FUNCTION_BLOCK "Blok_Jazdy_Band"	// FB 5
VERSION : 0.1
VAR
  Banda_1 : FB 30;
  Banda_2 : FB 30;
  Banda_3 : FB 30;
  Banda_4 : FB 31;
  Banda_5 : FB 30;
  Banda_6 : FB 30;
  Banda_7 : FB 30;
  Banda_8 : FB 30;
  Banda_9 : FB 30;
  Banda_12 : FB 30;
  Banda_13 : FB 32;
  Banda_14 : FB 30;
END_VAR
BEGIN
NETWORK
TITLE =
//Ten network celowo jest wolny
NETWORK
TITLE =
//Opoznienie wlotu bandy 1
//Uwaga Stare !!!
//      CALL  "Opoznienie_Wlotu"
//       Wejscie :="AIO".Banda_1.Foto_1
//       Timmer_1:=T12
//       Timmer_2:=T13
//       Wyjscie :="M_Foto_1_Banda_1"
//       Zmienna :="Help_M_40_3"
NETWORK
TITLE =
//Banda 1
//Uwaga Stare !!!
//      CALL  #Banda_1
//       S_Marka_Bezpieczenstwa :="Marka_Bezpieczenstwa"
//       i_Foto_Koniec          :="M_Foto_1_Banda_1"
//       i_Zez_Od_Nast          :="AIO".Banda_2.Zez_Do_Pop
//       i_Paleta_Dost_Od_Nast  :="AIO".Banda_2.Paleta_Dost_do_Pop
//       i_Zabierz_Od_Pop       :=
//       Czas_Kontroli_Przejazdu:=T#10S
//       o_Zabierz_Do_Nast      :="AIO".Banda_1.Zabierz_do_Nast
//       o_Zez_Do_Pop           :="AIO".Banda_1.Zez_Do_Pop
//       o_Paleta_Dost_do_Pop   :="AIO".Banda_1.Paleta_Dost_do_Pop
//       o_Motor_Lewo           :="AIO".Banda_1.C_Wise
NETWORK
TITLE =
//Banda 2. Uznawana za Wlot 1
//Uwaga Stare !!!
//      CALL  #Banda_2
//       S_Marka_Bezpieczenstwa :="Marka_Bezpieczenstwa"
//       i_Foto_Koniec          :="AIO".Banda_2.Foto_1
//       i_Zez_Od_Nast          :="AIO".Banda_4.Zez_Do_Pop_Wlot_1
//       i_Paleta_Dost_Od_Nast  :="AIO".Banda_4.Potw_Dost_Wlot_1
//       i_Zabierz_Od_Pop       :="AIO".Banda_1.Zabierz_do_Nast
//       Czas_Kontroli_Przejazdu:=T#10S
//       o_Zabierz_Do_Nast      :="AIO".Banda_2.Zabierz_do_Nast
//       o_Zez_Do_Pop           :="AIO".Banda_2.Zez_Do_Pop
//       o_Paleta_Dost_do_Pop   :="AIO".Banda_2.Paleta_Dost_do_Pop
//       o_Motor_Lewo           :="AIO".Banda_2.C_Wise
NETWORK
TITLE =
//Opoznienie wlotu banda 3
      CALL  "Opoznienie_Wlotu" (
           Wejscie                  := "AIO".Banda_3.Foto_1,
           Timmer_1                 := T 14,
           Timmer_2                 := T 15,
           Wyjscie                  := "M_Foto_1_Banda_3",
           Zmienna                  := "Help_M_40_5");
NETWORK
TITLE =
//Banda 3. Uznawana za Wlot 2
      CALL  #Banda_3 (
           S_Marka_Bezpieczenstwa   := "Marka_Bezpieczenstwa",
           i_Foto_Koniec            := "M_Foto_1_Banda_3",
           i_Zez_Od_Nast            := DIX 7.2,
           i_Paleta_Dost_Od_Nast    := DIX 7.3,
           Czas_Kontroli_Przejazdu  := T#10S,
           o_Zabierz_Do_Nast        := DIX 5.2,
           o_Zez_Do_Pop             := DIX 5.0,
           o_Paleta_Dost_do_Pop     := DIX 5.1,
           o_Motor_Lewo             := DIX 4.4);
NETWORK
TITLE =
//Banda 4 obrotowa
      CALL  #Banda_4 (
           i_Marka_bezpieczenstwa   := "Marka_Bezpieczenstwa",
           i_Foto_1                 := DIX 6.2,
           i_Foto_2                 := DIX 6.3,
           i_Zez_od_Nast            := DIX 9.0,
           i_Zabierz_od_Wlot_1      := DIX 3.2,
           i_Zabierz_od_Wlot_2      := DIX 5.2,
           i_Paleta_Odb_Wylot       := DIX 9.1,
           i_czuj_poz_Wlot_1        := DIX 36.3,
           i_czuj_ham_Wlot_1        := DIX 36.2,
           i_czuj_poz_Wlot_2        := DIX 36.0,
           i_czuj_ham_Wlot_2        := DIX 36.1,
           i_Foto_Wlot_1            := "M_Foto_1_Banda_2",
           i_Foto_Wlot_2            := "M_Foto_1_Banda_3",
           o_Zez_do_Wlot_1          := DIX 7.0,
           o_Zez_do_Wlot_2          := DIX 7.2,
           o_Paleta_Dost_Wlot_1     := DIX 7.1,
           o_Paleta_Dost_Wlot_2     := DIX 7.3,
           o_Zabierz_do_Nast        := DIX 7.4,
           o_Motor_1_lewo           := DIX 6.4,
           o_Motor_1_prawo          := DIX 6.5,
           o_Motor_2_obr_s_Wlot_1   := DIX 34.5,
           o_Motor_2_obr_s_Wlot_2   := DIX 34.4,
           o_Motor_2_Wolno          := DIX 34.6);
NETWORK
TITLE =
//Banda 5
      CALL  #Banda_5 (
           S_Marka_Bezpieczenstwa   := "Marka_Bezpieczenstwa",
           i_Foto_Koniec            := DIX 8.2,
           i_Zez_Od_Nast            := DIX 11.0,
           i_Paleta_Dost_Od_Nast    := DIX 11.1,
           i_Zabierz_Od_Pop         := DIX 7.4,
           Czas_Kontroli_Przejazdu  := T#10S,
           o_Zabierz_Do_Nast        := DIX 9.2,
           o_Zez_Do_Pop             := DIX 9.0,
           o_Paleta_Dost_do_Pop     := DIX 9.1,
           o_Motor_Lewo             := DIX 8.4);
NETWORK
TITLE =
//Banda 6
      CALL  #Banda_6 (
           S_Marka_Bezpieczenstwa   := "Marka_Bezpieczenstwa",
           i_Foto_Koniec            := DIX 10.2,
           i_Zez_Od_Nast            := DIX 13.0,
           i_Paleta_Dost_Od_Nast    := DIX 13.1,
           i_Zabierz_Od_Pop         := DIX 9.2,
           Czas_Kontroli_Przejazdu  := T#10S,
           o_Zabierz_Do_Nast        := DIX 11.2,
           o_Zez_Do_Pop             := DIX 11.0,
           o_Paleta_Dost_do_Pop     := DIX 11.1,
           o_Motor_Lewo             := DIX 10.4);
NETWORK
TITLE =
//Banda 7
      CALL  #Banda_7 (
           S_Marka_Bezpieczenstwa   := "Marka_Bezpieczenstwa",
           i_Foto_Koniec            := DIX 12.2,
           i_Zez_Od_Nast            := DIX 15.0,
           i_Paleta_Dost_Od_Nast    := DIX 15.1,
           i_Zabierz_Od_Pop         := DIX 11.2,
           Czas_Kontroli_Przejazdu  := T#10S,
           o_Zabierz_Do_Nast        := DIX 13.2,
           o_Zez_Do_Pop             := DIX 13.0,
           o_Paleta_Dost_do_Pop     := DIX 13.1,
           o_Motor_Lewo             := DIX 12.4);
NETWORK
TITLE =
//Banda 8
      CALL  #Banda_8 (
           S_Marka_Bezpieczenstwa   := "Marka_Bezpieczenstwa",
           i_Foto_Koniec            := DIX 14.2,
           i_Zez_Od_Nast            := DIX 17.0,
           i_Paleta_Dost_Od_Nast    := DIX 17.1,
           i_Zabierz_Od_Pop         := DIX 13.2,
           Czas_Kontroli_Przejazdu  := T#10S,
           o_Zabierz_Do_Nast        := DIX 15.2,
           o_Zez_Do_Pop             := DIX 15.0,
           o_Paleta_Dost_do_Pop     := DIX 15.1,
           o_Motor_Lewo             := DIX 14.4);
NETWORK
TITLE =
//Banda 9
      CALL  #Banda_9 (
           S_Marka_Bezpieczenstwa   := "Marka_Bezpieczenstwa",
           i_Foto_Koniec            := DIX 16.2,
           i_Zez_Od_Nast            := DIX 19.0,
           i_Paleta_Dost_Od_Nast    := DIX 19.1,
           i_Zabierz_Od_Pop         := DIX 15.2,
           Czas_Kontroli_Przejazdu  := T#10S,
           o_Zabierz_Do_Nast        := DIX 17.2,
           o_Zez_Do_Pop             := DIX 17.0,
           o_Paleta_Dost_do_Pop     := DIX 17.1,
           o_Motor_Lewo             := DIX 16.4);
NETWORK
TITLE = Zezwolenie do poprzedniej
//Banda 10 to foliarka. Tu jest interface laczacy dwie maszyny
      A     "MPI_GD".IN.Zezwolenie_Na_Wjazd_10;
      =     "AIO".Banda_10.Zez_Do_Pop;
//---
      A     "MPI_GD".IN.Potw_Dost_Na_Wjazd_10;
      =     "AIO".Banda_10.Paleta_Dost_do_Pop;
      A     "AIO".Banda_9.Zabierz_do_Nast;
      =     "MPI_GD".OUT.Zabierz_Na_Bande_10;
NETWORK
TITLE =
//Banda 11 to wylot z foliarki. Tu jest interface laczacy.Uwazana jako wlot 1
      A     "AIO".Banda_13.Zez_Do_Pop_Wlot_1;
      =     "MPI_GD".OUT.Zezwolenie_Na_Wyjazd_11;
//Przedluzenine czasu trwania sygnalu potwierdzenia
      A     "AIO".Banda_13.Potw_Dost_Wlot_1;
      L     S5T#200MS;
      SE    T 20;
      A     T 20;
      =     "MPI_GD".OUT.Potw_Dost_Na_Wyjazd_11;
//Przejecie palety
      A     "MPI_GD".IN.Zabierz_Na_Bande_11;
      =     "AIO".Banda_11.Zabierz_do_Nast;
      A     "MPI_GD".IN.Paleta_Obecna_Na_7_Tr;
      =     "M_Foto_1_Banda_11";
      A     "AIO".Czuj_21.Czujnik_90_St;
      AN    "AIO".Czuj_21.Czujnik_0_St;
      AN    "AIO".Czuj_22.Czujnik_45_St_CW;
      AN    "AIO".Czuj_22.Czujnik_45_St_CCW;
      =     "MPI_GD".OUT.Obrot_Na_Poz_Wlot_1;
NETWORK
TITLE =
//Opoznienie wlotu 2 przy obrotnicy 2
      CALL  "Opoznienie_Wlotu" (
           Wejscie                  := "AIO".Banda_12.Foto_1,
           Timmer_1                 := T 16,
           Timmer_2                 := T 17,
           Wyjscie                  := "M_Foto_1_Banda_12",
           Zmienna                  := "Help_M_40_7");
NETWORK
TITLE =
//Banda 12. Uwazana jako wlot 2.
      CALL  #Banda_12 (
           S_Marka_Bezpieczenstwa   := "Marka_Bezpieczenstwa",
           i_Foto_Koniec            := "M_Foto_1_Banda_12",
           i_Zez_Od_Nast            := DIX 25.2,
           i_Paleta_Dost_Od_Nast    := DIX 25.3,
           Czas_Kontroli_Przejazdu  := T#10S,
           o_Zabierz_Do_Nast        := DIX 23.2,
           o_Zez_Do_Pop             := DIX 23.0,
           o_Paleta_Dost_do_Pop     := DIX 23.1,
           o_Motor_Lewo             := DIX 22.4);
NETWORK
TITLE =
//banda 13 obrotowa
      CALL  #Banda_13 (
           i_Marka_bezpieczenstwa   := "Marka_Bezpieczenstwa",
           i_Foto_1                 := DIX 24.2,
           i_Foto_2                 := DIX 24.3,
           i_Zez_od_Nast            := DIX 27.0,
           i_Zabierz_od_Wlot_1      := DIX 21.2,
           i_Zabierz_od_Wlot_2      := DIX 23.2,
           i_Paleta_Odb_Wylot       := DIX 27.1,
           i_czuj_poz_Wlot_1        := DIX 40.3,
           i_czuj_ham_Wlot_1        := DIX 40.2,
           i_czuj_poz_Wlot_2        := DIX 40.0,
           i_czuj_ham_Wlot_2        := DIX 40.1,
           i_Czuj_poz_45_deg        := DIX 42.0,
           i_Czuj_ham_45_deg        := DIX 42.1,
           i_Foto_Wlot_1            := "M_Foto_1_Banda_11",
           i_Foto_Wlot_2            := "M_Foto_1_Banda_12",
           i_Etyk_praca_wlacz       := "Praca_Z_Etykietami",
           i_Etyk_poz_podst         := "Silownik_Etyk_Tyl",
           i_Etyk_obraz_w_pamieci   := "Dane_W_Drukarce",
           i_Etyk_syg_gotowosci     := "Etyk_Gotowa",
           i_Etyk_brak_materialu    := "Brak_Papieru",
           i_Etyk_Przycisk_Drukuj   := "Drukuj_Recznie",
           o_Zez_do_Wlot_1          := DIX 25.0,
           o_Zez_do_Wlot_2          := DIX 25.2,
           o_Paleta_Dost_Wlot_1     := DIX 25.1,
           o_Paleta_Dost_Wlot_2     := DIX 25.3,
           o_Zabierz_do_Nast        := DIX 25.4,
           o_Motor_1_lewo           := DIX 24.4,
           o_Motor_1_prawo          := DIX 24.5,
           o_Motor_2_obr_s_Wlot_1   := DIX 38.5,
           o_Motor_2_obr_s_Wlot_2   := DIX 38.4,
           o_Motor_2_Wolno          := DIX 38.6,
           o_Silownik_etykiety      := "Silownik_Etykiet",
           o_Drukuj_Etykiete        := "Drukuj_Etykiete",
           o_Zalaczenie_Skanera     := "Zalacz_Skaner",
           o_Lampka_Przycisk_Drukuj := "Lampka_Obraz_W_Pamieci");
NETWORK
TITLE =
//Wywolanie opoznienia zatrzymania fotokomorki po wyjsciu z obrotnicy
      CALL  "Opoznienie_Wylotu" (
           Wejscie                  := "AIO".Banda_14.Foto_1,
           Timmer_1                 := T 10,
           Timmer_2                 := T 11,
           Wyjscie                  := "M_Foto_1_Banda_14",
           Zmienna                  := "Help_M_40_1");
NETWORK
TITLE =
//Banda 14.Banda uwazana jako wylot z obrotnicy.
      CALL  #Banda_14 (
           S_Marka_Bezpieczenstwa   := "Marka_Bezpieczenstwa",
           i_Foto_Koniec            := "M_Foto_1_Banda_14",
           i_Zabierz_Od_Pop         := DIX 25.4,
           Czas_Kontroli_Przejazdu  := T#10S,
           o_Zabierz_Do_Nast        := DIX 27.2,
           o_Zez_Do_Pop             := DIX 27.0,
           o_Paleta_Dost_do_Pop     := DIX 27.1,
           o_Motor_Lewo             := DIX 26.4);
//      SET   
//      S     "Zalacz_Skaner"
END_FUNCTION_BLOCK

FUNCTION_BLOCK "Filtr_zbocza_2"	// FB 14
//Funkcja wykrywajace zbocze fotokomorki uwzgledniajaca nieczu³osc elementu
//
AUTHOR : Kng
FAMILY : Fun
NAME : Zb_1
VERSION : 0.1
VAR_INPUT
  Foto : BOOL ;
END_VAR
VAR_OUTPUT
  pos_zbocze : BOOL ;
END_VAR
VAR
  Opoz_zbocza_pos : SFB 4;
  p_Sygnal_foto : BOOL ;
  b_Opoz_poz : BOOL ;
  Help_zb_poz : BOOL ;
END_VAR
BEGIN
NETWORK
TITLE =
      CALL  #Opoz_zbocza_pos (
           IN                       := #Foto,
           PT                       := T#100MS,
           Q                        := #b_Opoz_poz);
      A     #b_Opoz_poz;
      S     #p_Sygnal_foto;
      AN    #Foto;
      R     #p_Sygnal_foto;
      A     #p_Sygnal_foto;
      FP    #Help_zb_poz;
      =     #pos_zbocze;
      BEU;
END_FUNCTION_BLOCK

FUNCTION_BLOCK "T_ON"	// FB 20
//Funkcja zatrzymujaca czas gdy na wejsciu stop pojawi sie stan niski. Wartosc 
//wejscia TON nie jest wtedy brana pod uwage. 
AUTHOR : Kng
NAME : Help_FB
VERSION : 0.1
VAR_INPUT
  IN : BOOL ;	//Wejscie aktywujace timer
  STOP : BOOL ;	//Sygnal aktywny stanem wysokim
  PT : TIME ;	//Czas zadany
END_VAR
VAR_OUTPUT
  Q_0 : BOOL ;
END_VAR
VAR_IN_OUT
  ET : TIME ;
END_VAR
VAR
  T_1 : SFB 4;
  Help_Zbocze_1 : BOOL ;
  Help_Zbocze_2 : BOOL ;
  Help_Zbocze_3 : BOOL ;
END_VAR
BEGIN
NETWORK
TITLE =
//Ten network celowo jest wolny
NETWORK
TITLE =
// Zapisanie wartosci czasu w pamieci
      A     #STOP;
      FN    #Help_Zbocze_1;
      A     #IN;
      JCN   et_1;
      L     #T_1.PT;
      L     #T_1.ET;
      -D;
      T     #T_1.PT;
      SET;
      R     #T_1.IN;
et_1: NOP   0;
//Przywrocenie czasu zapisanego
      A     #STOP;
      FP    #Help_Zbocze_2;
      A     #IN;
      S     #T_1.IN;
//Warunki poczatkowe
      A     #IN;
      FP    #Help_Zbocze_3;
      A     #STOP;
      JCN   et_3;
      L     #PT;
      T     #T_1.PT;
      SET;
      S     #T_1.IN;
et_3: NOP   0;
//Wywolaj funkcje timera
      CALL  #T_1;
      A     #T_1.Q;
      S     #Q_0;
      AN    #IN;
      A     #STOP;
//Wystaw wyjscie gdy skonczy sie czas
      R     #T_1.IN;
      R     #Q_0;
      L     #T_1.PT;
      L     #T_1.ET;
      -D;
      T     #ET;
//Pokaz wartosc czasu
END_FUNCTION_BLOCK

FUNCTION_BLOCK "T_ON_+_RESET"	// FB 21
//Funkcja zatrzymujaca czas gdy na wejsciu stop pojawi sie stan niski. Wartosc 
//wejscia TON nie jest wtedy brana pod uwage. 
//Dodano przycisk reset.
AUTHOR : Kng
NAME : Help_FB
VERSION : 1.1
VAR_INPUT
  IN : BOOL ;	//Wejscie aktywujace timer
  STOP : BOOL ;	//Sygnal aktywny stanem wysokim
  PT : TIME ;	//Czas zadany
  RESET : BOOL ;	//Wejescie resetujace aktywne stanem wysokim
END_VAR
VAR_OUTPUT
  Q_0 : BOOL ;
END_VAR
VAR_IN_OUT
  ET : TIME ;
END_VAR
VAR
  T_1 : SFB 4;
  Help_Zbocze_1 : BOOL ;
  Help_Zbocze_2 : BOOL ;
  Help_Zbocze_3 : BOOL ;
  Help_Zbocze_4 : BOOL ;
  Help_Zbocze_5 : BOOL ;
END_VAR
BEGIN
NETWORK
TITLE =
//Ten network celowo jest wolny
NETWORK
TITLE =
      A     #RESET;
      S     #Help_Zbocze_4;
// Zapisanie wartosci czasu w pamieci
      A     #STOP;
      FN    #Help_Zbocze_1;
      A     #IN;
      JCN   et_2;
      L     #T_1.PT;
      L     #T_1.ET;
      -D;
      T     #T_1.PT;
      SET;
      R     #T_1.IN;
et_2: NOP   0;
//Przywrocenie czasu zapisanego
      A     #STOP;
      FP    #Help_Zbocze_2;
      A     #IN;
      S     #T_1.IN;
//Wystaw wyjscie gdy skonczy sie czas
      A     #T_1.Q;
      S     #Q_0;
      AN    #IN;
      A     #STOP;
      O;
      A     #RESET;
      R     #T_1.IN;
      R     #Q_0;
//Warunki poczatkowe  oraz reset
      AN    #RESET;
      A     #Help_Zbocze_4;
      O;
      A(;
      A     #IN;
      FP    #Help_Zbocze_3;
      A     #STOP;
      );
      JCN   et_3;
      L     #PT;
      T     #T_1.PT;
      SET;
      R     #Help_Zbocze_4;
//brak wysterownia jezeli reset robiony bez stopu
      A     #STOP;
      S     #T_1.IN;
et_3: NOP   0;
//Wywolaj funkcje timera
      CALL  #T_1;
      L     #T_1.PT;
      L     #T_1.ET;
      -D;
      T     #ET;
//Pokaz wartosc czasu
END_FUNCTION_BLOCK

FUNCTION_BLOCK "Banda_Podwojna"	// FB 29
//Funkcja realizujaca koncepcje bandy podwojnej:
//-pojedynczy silnik
//-2 fotokomorki
//
AUTHOR : Kng
FAMILY : Bandy
NAME : B_dual
VERSION : 0.3
VAR_INPUT
  S_Marka_Bezpieczenstwa : BOOL ;
  i_Foto_Srodek : BOOL ;	//Foto na srodku tasmy
  i_Foto_Koniec : BOOL ;	//Foto na koncu tasmy
  i_Zez_Od_Nast : BOOL ;
  i_Paleta_Dost_Od_Nast : BOOL ;
  i_Zabierz_Od_Pop : BOOL ;
  Czas_Kontroli_Przejazdu : TIME ;
END_VAR
VAR_OUTPUT
  o_Zabierz_Do_Nast : BOOL ;	//Rozkaz pobrania do nast bandy
  o_Zez_Do_Pop : BOOL ;
  o_Paleta_Dost_do_Pop : BOOL ;
  o_Motor_Lewo : BOOL ;
END_VAR
VAR
  Czas_kontrolny : FB 20;
  Czas_Przejazdu : SFB 4;
  Help_Motor_Lewo : BOOL ;
  S_Dojazd_Po_Odebraniu : BOOL ;
  S_Help_Zab_Od_Pop : BOOL ;
  Stop_Czas_Kontrolny : BOOL ;
  Zbocze_1 : BOOL ;
  Zbocze_2 : BOOL ;
  Help_4 : BOOL ;
  Help_5 : BOOL ;
  Help_6 : BOOL ;
  Help_7 : BOOL ;
  Help_8 : BOOL ;
END_VAR
VAR_TEMP
  Temp_Help_1 : BOOL ;
  Temp_Help_2 : BOOL ;
  Czas_zadany : TIME ;
  Czas_aktualny : TIME ;
END_VAR
BEGIN
NETWORK
TITLE =
//
// B1        B2         foto_1    foto_2       B5        B6
//(\\\\\\\\\\\\\\\\\\)  (\\\\\\\\\\\\\\\\\\)  (\\\\\\\\\\\\\\\\\\)
//                  M1                    M2                     M3
//         
//        zabierz <-- pobierz      |  zabierz    <--  pobierz  
//     zez_do_pop --> zez_od_nast  |  zez_od_pop -->  zez_od_nast
//                                  
//-Uklad dzielony jest na realizowane funkcje
//
//         <----------------------------------------- kierunek
//                  
//
// ten network celowo jest pusty
NETWORK
TITLE =
      A     #S_Marka_Bezpieczenstwa;
      S     #Stop_Czas_Kontrolny;
NETWORK
TITLE =
//Wyznczenie zbocza pozytywnego i negatywnego
//Skocz jezeli brak marki bezpieczenstwa
      AN    #S_Marka_Bezpieczenstwa;
      AN    #Stop_Czas_Kontrolny;
      JC    end;
      AN    #S_Marka_Bezpieczenstwa;
      R     #Stop_Czas_Kontrolny;
NETWORK
TITLE =
// Opis poszczegolnych krokow i skok do nich
// Tasma poprzednia pusta i bierzaca pusta
      AN    #i_Foto_Koniec;
      AN    #o_Zabierz_Do_Nast;
      AN    #Help_Motor_Lewo;
      S     #o_Zez_Do_Pop;
      A     #i_Zabierz_Od_Pop;
      S     #Help_Motor_Lewo;
//Warunek gdy pobranie z poprzedniej i miejsce foto srodek
//jest zajete
      A     #i_Foto_Srodek;
      A     #i_Zabierz_Od_Pop;
      S     #S_Help_Zab_Od_Pop;
      A     #Help_Motor_Lewo;
      AN    #i_Zabierz_Od_Pop;
      =     #Temp_Help_1;
      CALL  #Czas_kontrolny (
           IN                       := #Temp_Help_1,
           STOP                     := #Stop_Czas_Kontrolny,
           PT                       := #Czas_Kontroli_Przejazdu,
           Q_0                      := #Temp_Help_2,
           ET                       := #Czas_aktualny);
//Paleta dostarczona
      A     #Temp_Help_2;
      O;
      A     #i_Foto_Koniec;
      FP    #Zbocze_2;
      O(;
      A     #i_Foto_Srodek;	//tu musi byc zbocze
      FP    #Zbocze_1;
      AN    #S_Help_Zab_Od_Pop;
      );
      R     #Help_Motor_Lewo;
      R     #S_Help_Zab_Od_Pop;
      R     #o_Zez_Do_Pop;
      =     #o_Paleta_Dost_do_Pop;
// foto srodek zajete, foto koniec ,zezwolenie od nastepnej;
//robione jest przejscie z jednej czesci bandy do drugiej
//nieaktualne dla 1 foto
      AN    #i_Foto_Koniec;
      A     #i_Foto_Srodek;
      A     #i_Zez_Od_Nast;
      S     #Help_Motor_Lewo;
//Wyjazd z drugiej czesci bandy
//jest zezwolenie od nastepnej
      A     #i_Foto_Koniec;
      A     #i_Zez_Od_Nast;
      S     #Help_Motor_Lewo;
      =     #o_Zabierz_Do_Nast;
      A     #i_Paleta_Dost_Od_Nast;
      S     #S_Dojazd_Po_Odebraniu;
      CALL  #Czas_Przejazdu (
           IN                       := #S_Dojazd_Po_Odebraniu,
           PT                       := T#100MS,
           Q                        := #Temp_Help_2,
           ET                       := #Czas_aktualny);
      A     #Temp_Help_2;
      O;
      A     #S_Dojazd_Po_Odebraniu;
      A     #i_Foto_Koniec;
      R     #Help_Motor_Lewo;
      R     #S_Dojazd_Po_Odebraniu;
//Gdy zajete Foto_1 brak zezwolenia do poprzedniej
      A     #i_Foto_Koniec;
      R     #o_Zez_Do_Pop;
//warunkowe zakonczenie pracy silnika gdy brak zezwolenia
//z nastepnej
      A     #i_Foto_Koniec;
      AN    #i_Zez_Od_Nast;
      R     #Help_Motor_Lewo;
NETWORK
TITLE =
end:  NOP   0;
      A     #S_Marka_Bezpieczenstwa;
      A     #Help_Motor_Lewo;
      =     #o_Motor_Lewo;
      BEU;
NETWORK
TITLE =
END_FUNCTION_BLOCK

FUNCTION_BLOCK "Banda_Pojedyncza"	// FB 30
//Funkcja realizujaca koncepcje bandy podwojnej:
//-pojedynczy silnik
//-2 fotokomorki
//
AUTHOR : Kng
FAMILY : Bandy
NAME : B_dual
VERSION : 0.0
VAR_INPUT
  S_Marka_Bezpieczenstwa : BOOL ;
  i_Foto_Koniec : BOOL ;	//Foto na koncu tasmy
  i_Zez_Od_Nast : BOOL ;
  i_Paleta_Dost_Od_Nast : BOOL ;
  i_Zabierz_Od_Pop : BOOL ;
  Czas_Kontroli_Przejazdu : TIME ;
END_VAR
VAR_OUTPUT
  o_Zabierz_Do_Nast : BOOL ;	//Rozkaz pobrania do nast bandy
  o_Zez_Do_Pop : BOOL ;
  o_Paleta_Dost_do_Pop : BOOL ;
  o_Motor_Lewo : BOOL ;
END_VAR
VAR
  Czas_kontrolny : FB 20;
  Help_Motor_Lewo : BOOL ;
  S_Dojazd_Po_Odebraniu : BOOL ;
  S_Help_Zab_Od_Pop : BOOL ;
  Stop_Czas_Kontrolny : BOOL ;
  Zbocze_1 : BOOL ;
  Zbocze_2 : BOOL ;
  Blokada_Wjazd : BOOL ;
  Help_5 : BOOL ;
  Help_6 : BOOL ;
  Help_7 : BOOL ;
  Help_8 : BOOL ;
END_VAR
VAR_TEMP
  Temp_Help_1 : BOOL ;
  Temp_Help_2 : BOOL ;
  Czas_zadany : TIME ;
  Czas_aktualny : TIME ;
END_VAR
BEGIN
NETWORK
TITLE =
//
// B1        B2         foto_1    foto_2         B5        B6
//(\\\\\\\\\\\\\\\\\\)  (\\\\\\\\\\\\\\\\\\)  (\\\\\\\\\\\\\\\\\\)
//                  M1                    M2                     M3
//         
//        zabierz <-- pobierz      |  zabierz    <--  pobierz  
//     zez_do_pop --> zez_od_nast  |  zez_od_pop -->  zez_od_nast
//                                  
//-Uklad dzielony jest na realizowane funkcje
//
//         <----------------------------------------- kierunek
//                  
//
// ten network celowo jest pusty
NETWORK
TITLE =
      A     #S_Marka_Bezpieczenstwa;
      S     #Stop_Czas_Kontrolny;
NETWORK
TITLE =
//Wyznczenie zbocza pozytywnego i negatywnego
//Skocz jezeli brak marki bezpieczenstwa
      AN    #S_Marka_Bezpieczenstwa;
      AN    #Stop_Czas_Kontrolny;
      JC    end;
      AN    #S_Marka_Bezpieczenstwa;
      R     #Stop_Czas_Kontrolny;
NETWORK
TITLE =
// Opis poszczegolnych krokow i skok do nich
// Tasma poprzednia pusta i bierzaca pusta
      AN    #i_Foto_Koniec;
      AN    #o_Zabierz_Do_Nast;
      AN    #Help_Motor_Lewo;
      S     #o_Zez_Do_Pop;
      A     #i_Zabierz_Od_Pop;
      S     #Help_Motor_Lewo;
      S     #Blokada_Wjazd;
//Warunek gdy pobranie z poprzedniej i miejsce foto srodek
//jest zajete
      A     #Help_Motor_Lewo;
      AN    #i_Zabierz_Od_Pop;
      AN    #i_Foto_Koniec;
      =     #Temp_Help_1;
      CALL  #Czas_kontrolny (
           IN                       := #Temp_Help_1,
           STOP                     := #Stop_Czas_Kontrolny,
           PT                       := #Czas_Kontroli_Przejazdu,
           Q_0                      := #Temp_Help_2,
           ET                       := #Czas_aktualny);
//Paleta dostarczona
      A     #Temp_Help_2;
      O;
      A     #i_Foto_Koniec;
      FP    #Zbocze_2;
      R     #Help_Motor_Lewo;
      R     #o_Zez_Do_Pop;
      =     #o_Paleta_Dost_do_Pop;
//jest zezwolenie od nastepnej
      A     #i_Foto_Koniec;
      A     #i_Zez_Od_Nast;
      S     #Help_Motor_Lewo;
      =     #o_Zabierz_Do_Nast;
//Potwierdzenie otrzymania palety
      AN    #Blokada_Wjazd;
      A     #i_Paleta_Dost_Od_Nast;
      FP    #Zbocze_1;
      R     #Help_Motor_Lewo;
//Gdy zajete Foto_1 brak zezwolenia do poprzedniej
      A     #i_Foto_Koniec;
      R     #o_Zez_Do_Pop;
      R     #Blokada_Wjazd;
//warunkowe zakonczenie pracy silnika gdy brak zezwolenia
//z nastepnej
      A     #i_Foto_Koniec;
      AN    #i_Zez_Od_Nast;
      R     #Help_Motor_Lewo;
NETWORK
TITLE =
end:  NOP   0;
      A     #S_Marka_Bezpieczenstwa;
      A     #Help_Motor_Lewo;
      =     #o_Motor_Lewo;
      BEU;
NETWORK
TITLE =
END_FUNCTION_BLOCK

FUNCTION_BLOCK "Banda_Obr_1"	// FB 31
AUTHOR : Kng
FAMILY : Bandy
NAME : Band_obr
VERSION : 0.1
VAR_INPUT
  i_Marka_bezpieczenstwa : BOOL ;
  i_Foto_1 : BOOL ;
  i_Foto_2 : BOOL ;
  i_Zez_od_Nast : BOOL ;
  i_Zabierz_od_Wlot_1 : BOOL ;
  i_Zabierz_od_Wlot_2 : BOOL ;
  i_Paleta_Odb_Wylot : BOOL ;
  i_czuj_poz_Wlot_1 : BOOL ;
  i_czuj_ham_Wlot_1 : BOOL ;
  i_czuj_poz_Wlot_2 : BOOL ;
  i_czuj_ham_Wlot_2 : BOOL ;
  i_Foto_Wlot_1 : BOOL ;
  i_Foto_Wlot_2 : BOOL ;
END_VAR
VAR_OUTPUT
  o_Zez_do_Wlot_1 : BOOL ;
  o_Zez_do_Wlot_2 : BOOL ;
  o_Paleta_Dost_Wlot_1 : BOOL ;
  o_Paleta_Dost_Wlot_2 : BOOL ;
  o_Zabierz_do_Nast : BOOL ;
  o_Motor_1_lewo : BOOL ;
  o_Motor_1_prawo : BOOL ;
  o_Motor_2_obr_s_Wlot_1 : BOOL ;	//Motor obrotnicy,kierunek strona wejscia,szybko
  o_Motor_2_obr_s_Wlot_2 : BOOL ;	//Motor obrotnicy,kierunek strona wyjscia,szybko
  o_Motor_2_Wolno : BOOL ;	//Motor obrotnicy,kierunek strona wejscia,wolno
END_VAR
VAR
  Kontrola_Rolki_Wlot_1 : FB 20;
  Dojazd_Rolki_Wlot_1 : FB 20;
  Kontrola_Rolki_Wlot_2 : FB 20;
  Dojazd_Rolki_Wlot_2 : FB 20;
  Czas_kontrolny : SFB 4;	//Czas kontrolny wjazdu palety
  Sterownie_Obrotnicy : FB 51;
  Opuszczenie_Bandy : SFB 4;
  Silniki_nie_pracuja : BOOL ;
  Help_Motor_1_lewo : BOOL ;
  Help_Motor_1_prawo : BOOL ;
  Help_Motor_2_obr_Wlot_1 : BOOL ;	//Motor obrotnicy,kierunek strona wejscia,szybko
  Help_Motor_2_obr_Wlot_2 : BOOL ;	//Motor obrotnicy,kierunek strona wyjscia,szybko
  Help_Motor_2_Wolno : BOOL ;	//Motor obrotnicy,kierunek strona wejscia,wolno
  Blokada_Na_Wlot_1 : BOOL ;
  Blokada_Na_Wlot_2 : BOOL ;
  Blokada_Wlotu : BOOL ;
  Poz_Wlot_1 : BOOL ;
  Poz_Wlot_2 : BOOL ;
  Obr_Na_Wlot_1 : BOOL ;
  Obr_Na_wlot_2 : BOOL ;
  Odblokuj_Obrotnice : BOOL ;
  Rolki_Odblokowane : BOOL ;
  Stop_Czas_Kontrolny : BOOL ;
  Filtr_Rolki_Wlot_1 : BOOL ;
  H1_Doj_Rolki_Wlot_1 : BOOL ;
  H2_Doj_Rolki_Wlot_1 : BOOL ;
  Filtr_Rolki_Wlot_2 : BOOL ;
  H1_Doj_Rolki_Wlot_2 : BOOL ;
  H2_Doj_Rolki_Wlot_2 : BOOL ;
  Pobranie_Wlot_1 : BOOL ;
  Pobranie_Wlot_2 : BOOL ;
  Paleta_Na_Obrotnicy : BOOL ;
  Oddanie_Palety : BOOL ;
  Zbocze_1 : BOOL ;
  Zbocze_2 : BOOL ;
  Zbocze_3 : BOOL ;
  Wybor_Wjazdu : FB 50;
  Help_Zez_Wlot_1 : BOOL ;
  Help_Zez_Wlot_2 : BOOL ;
END_VAR
VAR_TEMP
  Temp_Help_1 : BOOL ;
  Temp_Help_2 : BOOL ;
  Czas_zadany : TIME ;
  Czas_aktualny : TIME ;
END_VAR
BEGIN
NETWORK
TITLE =
//                   
//Wlot 1                               Wylot
//()()()()|()()()()|  ()()()  |()()()()|()()()()
//()()()()|()()()()| ()()()() |()()()()|()()()()
//()()()()|()()()()| ()()()() |()()()()|()()()()
//()()()()|()()()()| ()()()() |()()()()|()()()()
//()()()()|()()()()|  ()()()  |()()()()|()()()()
//
//                  |()()()()|
//                  |()()()()|
//                  |()()()()| 
//                  |()()()()|
//                    Wlot_2
//         
//          pobierz --> zabierz   |     pobierz --> zabierz   
//     zez_od_nast <-- zez_do_pop | zez_od_nast <-- zez_od_pop
//                                  
//-Uklad dzielony jest na realizowane funkcje
//
//         
//                  
//
// ten network celowo jest pusty
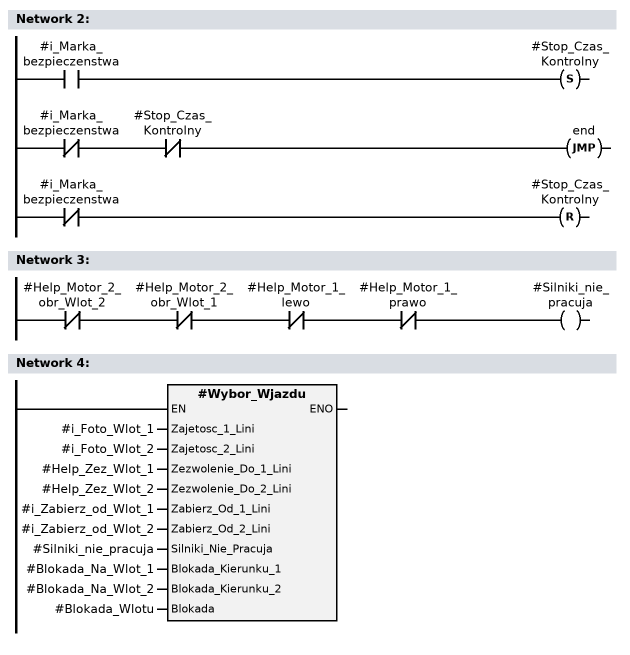
NETWORK
TITLE =
//Zatrzymanie uplywajacego czasu gdy brak bezpieczenstwa
//Skocz jezeli brak marki bezpieczenstwa
      A     #i_Marka_bezpieczenstwa;
      S     #Stop_Czas_Kontrolny;
      AN    #i_Marka_bezpieczenstwa;
      AN    #Stop_Czas_Kontrolny;
      JC    end;
      AN    #i_Marka_bezpieczenstwa;
      R     #Stop_Czas_Kontrolny;
NETWORK
TITLE =
//Sprawdzenie czy silniki nie pracuja
      AN    #Help_Motor_2_obr_Wlot_2;
      AN    #Help_Motor_2_obr_Wlot_1;
      AN    #Help_Motor_1_lewo;
      AN    #Help_Motor_1_prawo;
      =     #Silniki_nie_pracuja;
NETWORK
TITLE =
//Wybranie wjazdu
      CALL  #Wybor_Wjazdu (
           Zajetosc_1_Lini          := #i_Foto_Wlot_1,
           Zajetosc_2_Lini          := #i_Foto_Wlot_2,
           Zezwolenie_Do_1_Lini     := #Help_Zez_Wlot_1,
           Zezwolenie_Do_2_Lini     := #Help_Zez_Wlot_2,
           Zabierz_Od_1_Lini        := #i_Zabierz_od_Wlot_1,
           Zabierz_Od_2_Lini        := #i_Zabierz_od_Wlot_2,
           Silniki_Nie_Pracuja      := #Silniki_nie_pracuja,
           Blokada_Kierunku_1       := #Blokada_Na_Wlot_1,
           Blokada_Kierunku_2       := #Blokada_Na_Wlot_2,
           Blokada                  := #Blokada_Wlotu);
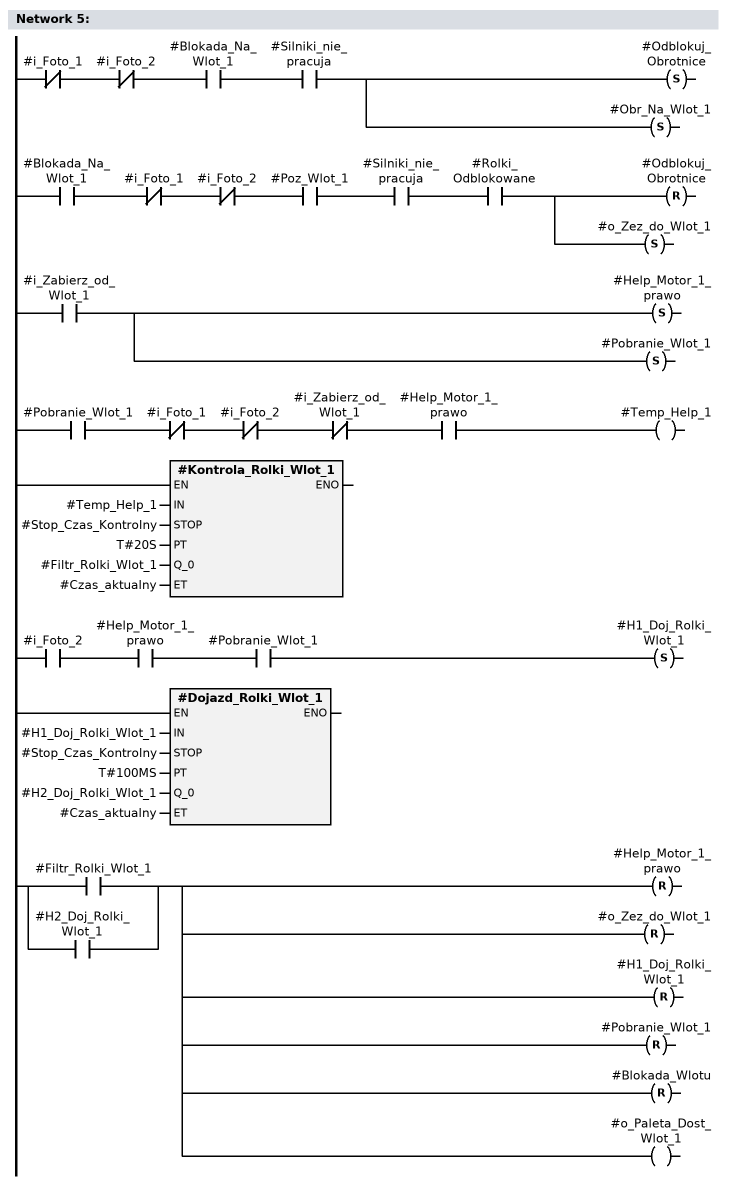
NETWORK
TITLE =
//Pobranie palety z Wlotu nr 1
//Obrot obrotnicy w kierunku wlotu nr 1
      AN    #i_Foto_1;
      AN    #i_Foto_2;
      A     #Blokada_Na_Wlot_1;
      A     #Silniki_nie_pracuja;
      S     #Odblokuj_Obrotnice;
      S     #Obr_Na_Wlot_1;
//Zezwolenie na wjazd z wlotu 1
      A     #Blokada_Na_Wlot_1;
      AN    #i_Foto_1;
      AN    #i_Foto_2;
      A     #Poz_Wlot_1;
      A     #Silniki_nie_pracuja;
      A     #Rolki_Odblokowane;
      R     #Odblokuj_Obrotnice;
      S     #o_Zez_do_Wlot_1;
//Gdy syganl zabierz to uruchom tasme
      A     #i_Zabierz_od_Wlot_1;
      S     #Help_Motor_1_prawo;
      S     #Pobranie_Wlot_1;
//Warunek gdy pobranie z poprzedniej i miejsce foto srodek
//jest zajete
      A     #Pobranie_Wlot_1;
      AN    #i_Foto_1;
      AN    #i_Foto_2;
      AN    #i_Zabierz_od_Wlot_1;
      A     #Help_Motor_1_prawo;
      =     #Temp_Help_1;
      CALL  #Kontrola_Rolki_Wlot_1 (
           IN                       := #Temp_Help_1,
           STOP                     := #Stop_Czas_Kontrolny,
           PT                       := T#20S,
           Q_0                      := #Filtr_Rolki_Wlot_1,
           ET                       := #Czas_aktualny);
      A     #i_Foto_2;
      A     #Help_Motor_1_prawo;
      A     #Pobranie_Wlot_1;
      S     #H1_Doj_Rolki_Wlot_1;
      CALL  #Dojazd_Rolki_Wlot_1 (
           IN                       := #H1_Doj_Rolki_Wlot_1,
           STOP                     := #Stop_Czas_Kontrolny,
           PT                       := T#100MS,
           Q_0                      := #H2_Doj_Rolki_Wlot_1,
           ET                       := #Czas_aktualny);
//Koniec pobierania palety z wlotu 1
      A     #Filtr_Rolki_Wlot_1;
      O;
      A     #H2_Doj_Rolki_Wlot_1;
      R     #Help_Motor_1_prawo;
      R     #o_Zez_do_Wlot_1;
      R     #H1_Doj_Rolki_Wlot_1;
      R     #Pobranie_Wlot_1;
      R     #Blokada_Wlotu;
      =     #o_Paleta_Dost_Wlot_1;
//-----------------------------------------------------
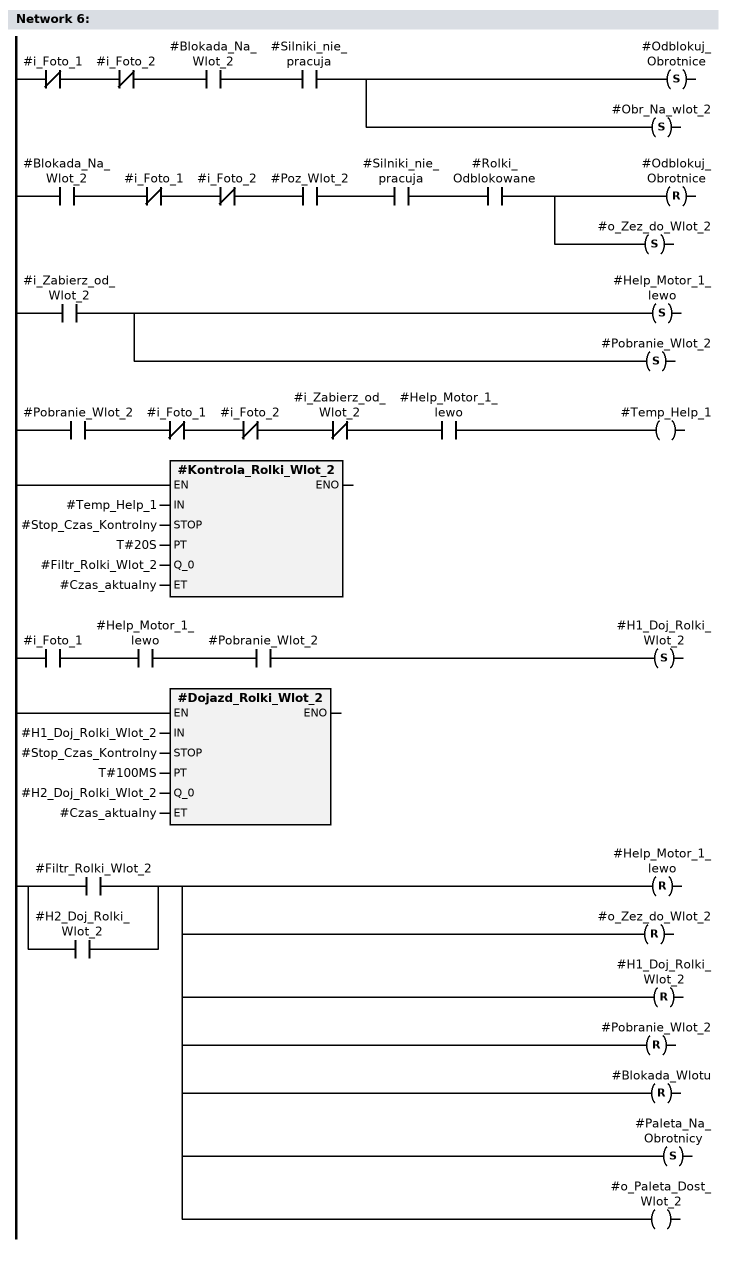
NETWORK
TITLE =
////Pobieranie Palety Wlot 2
//Obrot obrotnicy w kierunku wlotu nr 2
      AN    #i_Foto_1;
      AN    #i_Foto_2;
      A     #Blokada_Na_Wlot_2;
      A     #Silniki_nie_pracuja;
      S     #Odblokuj_Obrotnice;
      S     #Obr_Na_wlot_2;
//Zezwolenie na wjazd z wlotu 2
      A     #Blokada_Na_Wlot_2;
      AN    #i_Foto_1;
      AN    #i_Foto_2;
      A     #Poz_Wlot_2;
      A     #Silniki_nie_pracuja;
      A     #Rolki_Odblokowane;
      R     #Odblokuj_Obrotnice;
      S     #o_Zez_do_Wlot_2;
//Gdy syganl zabierz to uruchom tasme
      A     #i_Zabierz_od_Wlot_2;
      S     #Help_Motor_1_lewo;
      S     #Pobranie_Wlot_2;
//Warunek gdy pobranie z poprzedniej i miejsce foto srodek
//jest zajete
      A     #Pobranie_Wlot_2;
      AN    #i_Foto_1;
      AN    #i_Foto_2;
      AN    #i_Zabierz_od_Wlot_2;
      A     #Help_Motor_1_lewo;
      =     #Temp_Help_1;
      CALL  #Kontrola_Rolki_Wlot_2 (
           IN                       := #Temp_Help_1,
           STOP                     := #Stop_Czas_Kontrolny,
           PT                       := T#20S,
           Q_0                      := #Filtr_Rolki_Wlot_2,
           ET                       := #Czas_aktualny);
      A     #i_Foto_1;
      A     #Help_Motor_1_lewo;
      A     #Pobranie_Wlot_2;
      S     #H1_Doj_Rolki_Wlot_2;
      CALL  #Dojazd_Rolki_Wlot_2 (
           IN                       := #H1_Doj_Rolki_Wlot_2,
           STOP                     := #Stop_Czas_Kontrolny,
           PT                       := T#100MS,
           Q_0                      := #H2_Doj_Rolki_Wlot_2,
           ET                       := #Czas_aktualny);
//Koniec pobierania palety z wlotu 2
      A     #Filtr_Rolki_Wlot_2;
      O;
      A     #H2_Doj_Rolki_Wlot_2;
      R     #Help_Motor_1_lewo;
      R     #o_Zez_do_Wlot_2;
      R     #H1_Doj_Rolki_Wlot_2;
      R     #Pobranie_Wlot_2;
      R     #Blokada_Wlotu;
      S     #Paleta_Na_Obrotnicy;
      =     #o_Paleta_Dost_Wlot_2;
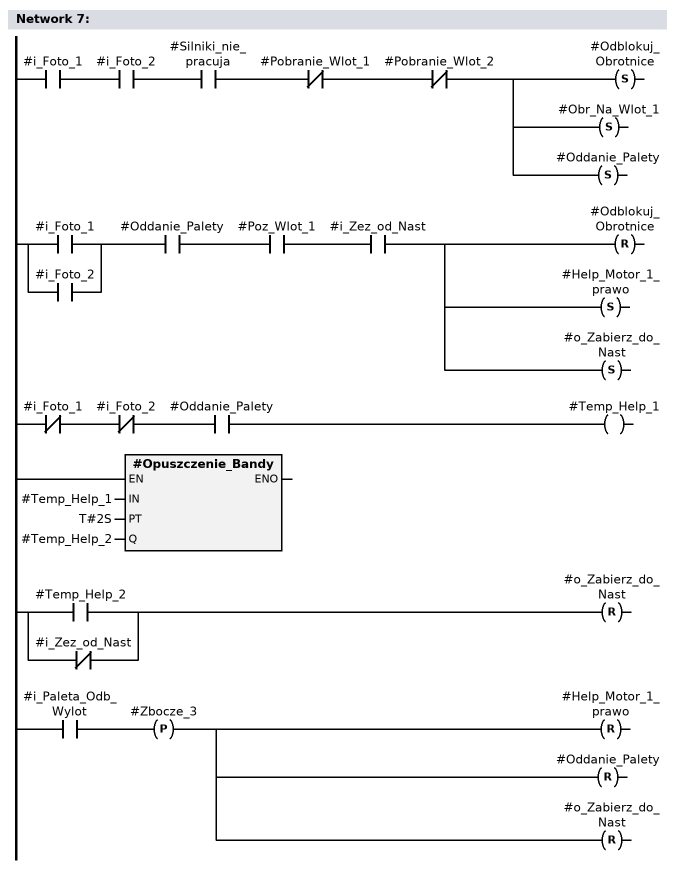
NETWORK
TITLE =
//Wyjazd palety z bandy obrotowej
      A     #i_Foto_1;
      A     #i_Foto_2;
      A     #Silniki_nie_pracuja;
      AN    #Pobranie_Wlot_1;
      AN    #Pobranie_Wlot_2;
      S     #Odblokuj_Obrotnice;
      S     #Obr_Na_Wlot_1;
      S     #Oddanie_Palety;
//Oczekiwanie na zezwolenie
      O     #i_Foto_1;
      O     #i_Foto_2;
      A     #Oddanie_Palety;
      A     #Poz_Wlot_1;
      A     #i_Zez_od_Nast;
      R     #Odblokuj_Obrotnice;
      S     #Help_Motor_1_prawo;
      S     #o_Zabierz_do_Nast;
//reset sygn³u zabierz
      AN    #i_Foto_1;
      AN    #i_Foto_2;
      A     #Oddanie_Palety;
      =     #Temp_Help_1;
      CALL  #Opuszczenie_Bandy (
           IN                       := #Temp_Help_1,
           PT                       := T#2S,
           Q                        := #Temp_Help_2);
      A     #Temp_Help_2;
      O;
      AN    #i_Zez_od_Nast;
      R     #o_Zabierz_do_Nast;
      A     #i_Paleta_Odb_Wylot;
      FP    #Zbocze_3;
      R     #Help_Motor_1_prawo;
      R     #Oddanie_Palety;
      R     #o_Zabierz_do_Nast;
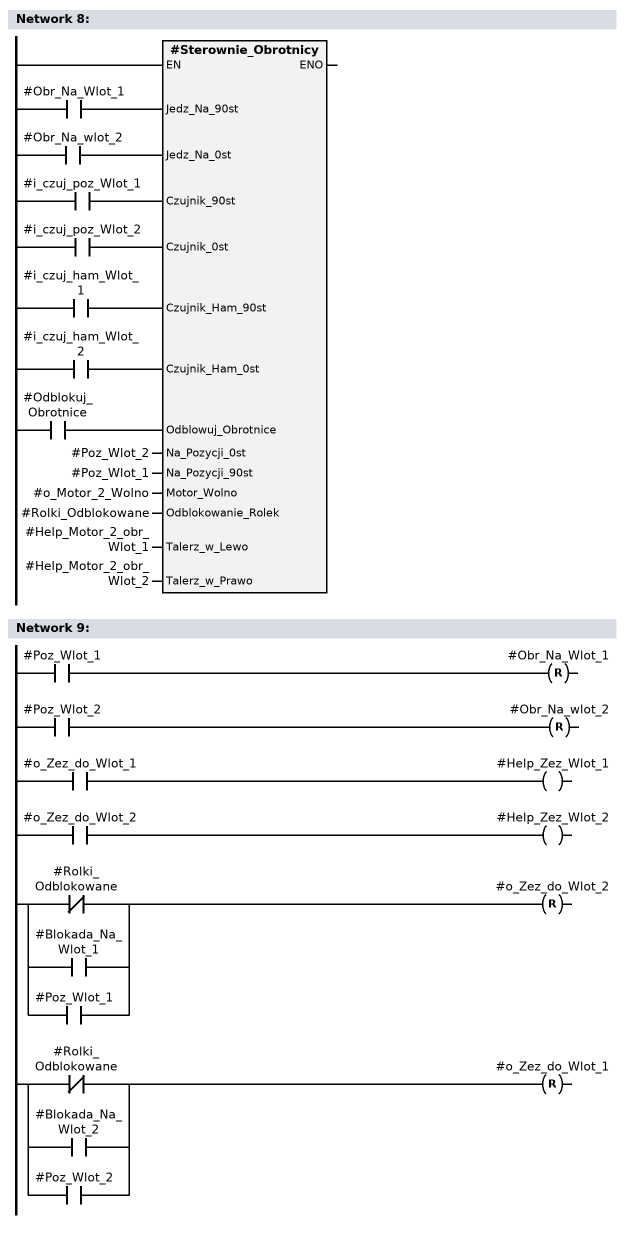
NETWORK
TITLE =
      A     #Obr_Na_Wlot_1;
      =     L 10.0;
      BLD   103;
      A     #Obr_Na_wlot_2;
      =     L 10.1;
      BLD   103;
      A     #i_czuj_poz_Wlot_1;
      =     L 10.2;
      BLD   103;
      A     #i_czuj_poz_Wlot_2;
      =     L 10.3;
      BLD   103;
      A     #i_czuj_ham_Wlot_1;
      =     L 10.4;
      BLD   103;
      A     #i_czuj_ham_Wlot_2;
      =     L 10.5;
      BLD   103;
      A     #Odblokuj_Obrotnice;
      =     L 10.6;
      BLD   103;
      CALL  #Sterownie_Obrotnicy (
           Jedz_Na_90st             := L 10.0,
           Jedz_Na_0st              := L 10.1,
           Czujnik_90st             := L 10.2,
           Czujnik_0st              := L 10.3,
           Czujnik_Ham_90st         := L 10.4,
           Czujnik_Ham_0st          := L 10.5,
           Odblowuj_Obrotnice       := L 10.6,
           Na_Pozycji_0st           := #Poz_Wlot_2,
           Na_Pozycji_90st          := #Poz_Wlot_1,
           Motor_Wolno              := #o_Motor_2_Wolno,
           Odblokowanie_Rolek       := #Rolki_Odblokowane,
           Talerz_w_Lewo            := #Help_Motor_2_obr_Wlot_1,
           Talerz_w_Prawo           := #Help_Motor_2_obr_Wlot_2);
      NOP   0;
NETWORK
TITLE =
//Warunki skrajne
      A     #Poz_Wlot_1;
      R     #Obr_Na_Wlot_1;
      A     #Poz_Wlot_2;
      R     #Obr_Na_wlot_2;
      A     #o_Zez_do_Wlot_1;
      =     #Help_Zez_Wlot_1;
      A     #o_Zez_do_Wlot_2;
      =     #Help_Zez_Wlot_2;
      ON    #Rolki_Odblokowane;
      O     #Blokada_Na_Wlot_1;
      O     #Poz_Wlot_1;
      R     #o_Zez_do_Wlot_2;
      ON    #Rolki_Odblokowane;
      O     #Blokada_Na_Wlot_2;
      O     #Poz_Wlot_2;
      R     #o_Zez_do_Wlot_1;
NETWORK
TITLE =
//Warunki skrajne
end:  NOP   0;
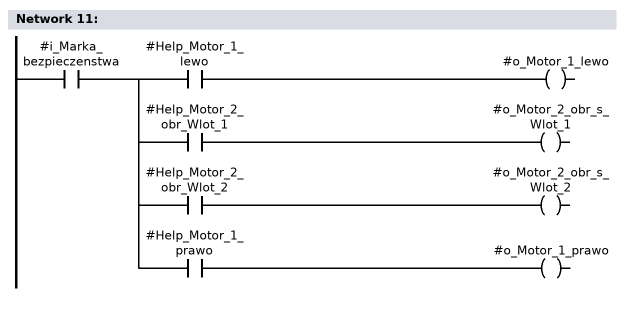
NETWORK
TITLE =
      A     #i_Marka_bezpieczenstwa;
      =     L 10.0;
      A     L 10.0;
      A     #Help_Motor_1_lewo;
      =     #o_Motor_1_lewo;
      A     L 10.0;
      A     #Help_Motor_2_obr_Wlot_1;
      =     #o_Motor_2_obr_s_Wlot_1;
      A     L 10.0;
      A     #Help_Motor_2_obr_Wlot_2;
      =     #o_Motor_2_obr_s_Wlot_2;
      A     L 10.0;
      A     #Help_Motor_1_prawo;
      =     #o_Motor_1_prawo;
NETWORK
TITLE =
END_FUNCTION_BLOCK

FUNCTION_BLOCK "Banda_Obr_2"	// FB 32
AUTHOR : Kng
FAMILY : Bandy
NAME : Band_obr
VERSION : 0.1
VAR_INPUT
  i_Marka_bezpieczenstwa : BOOL ;
  i_Foto_1 : BOOL ;
  i_Foto_2 : BOOL ;
  i_Zez_od_Nast : BOOL ;
  i_Zabierz_od_Wlot_1 : BOOL ;
  i_Zabierz_od_Wlot_2 : BOOL ;
  i_Paleta_Odb_Wylot : BOOL ;
  i_czuj_poz_Wlot_1 : BOOL ;
  i_czuj_ham_Wlot_1 : BOOL ;
  i_czuj_poz_Wlot_2 : BOOL ;
  i_czuj_ham_Wlot_2 : BOOL ;
  i_Czuj_poz_45_deg : BOOL ;
  i_Czuj_ham_45_deg : BOOL ;
  i_Foto_Wlot_1 : BOOL ;
  i_Foto_Wlot_2 : BOOL ;
  i_Etyk_praca_wlacz : BOOL ;
  i_Etyk_poz_podst : BOOL ;
  i_Etyk_obraz_w_pamieci : BOOL ;
  i_Etyk_syg_gotowosci : BOOL ;
  i_Etyk_brak_materialu : BOOL ;
  i_Etyk_Przycisk_Drukuj : BOOL ;
END_VAR
VAR_OUTPUT
  o_Zez_do_Wlot_1 : BOOL ;
  o_Zez_do_Wlot_2 : BOOL ;
  o_Paleta_Dost_Wlot_1 : BOOL ;
  o_Paleta_Dost_Wlot_2 : BOOL ;
  o_Zabierz_do_Nast : BOOL ;
  o_Motor_1_lewo : BOOL ;
  o_Motor_1_prawo : BOOL ;
  o_Motor_2_obr_s_Wlot_1 : BOOL ;	//Motor obrotnicy,kierunek strona wejscia,szybko
  o_Motor_2_obr_s_Wlot_2 : BOOL ;	//Motor obrotnicy,kierunek strona wyjscia,szybko
  o_Motor_2_Wolno : BOOL ;	//Motor obrotnicy,kierunek strona wejscia,wolno
  o_Silownik_etykiety : BOOL ;
  o_Drukuj_Etykiete : BOOL ;
  o_Zalaczenie_Skanera : BOOL ;
  o_Lampka_Przycisk_Drukuj : BOOL ;
END_VAR
VAR
  Kontrola_Rolki_Wlot_1 : FB 20;
  Dojazd_Rolki_Wlot_1 : FB 20;
  Kontrola_Rolki_Wlot_2 : FB 20;
  Dojazd_Rolki_Wlot_2 : FB 20;
  Czas_kontrolny : SFB 4;	//Czas kontrolny wjazdu palety
  Opuszczenie_Bandy : SFB 4;
  Wybor_Wjazdu : FB 50;
  Sterowanie_Obrotu : FB 52;
  Czas_Oczek_Na_Obraz : SFB 4;
  Silniki_nie_pracuja : BOOL ;
  Help_Motor_1_lewo : BOOL ;
  Help_Motor_1_prawo : BOOL ;
  Help_Motor_2_obr_Wlot_1 : BOOL ;	//Motor obrotnicy,kierunek strona wejscia,szybko
  Help_Motor_2_obr_Wlot_2 : BOOL ;	//Motor obrotnicy,kierunek strona wyjscia,szybko
  Help_Motor_2_Wolno : BOOL ;	//Motor obrotnicy,kierunek strona wejscia,wolno
  Blokada_Na_Wlot_1 : BOOL ;
  Blokada_Na_Wlot_2 : BOOL ;
  Blokada_Wlotu : BOOL ;
  Poz_Wlot_1 : BOOL ;
  Poz_Wlot_2 : BOOL ;
  Obr_Na_Wlot_1 : BOOL ;
  Obr_Na_wlot_2 : BOOL ;
  Odblokuj_Obrotnice : BOOL ;
  Rolki_Odblokowane : BOOL ;
  Stop_Czas_Kontrolny : BOOL ;
  Filtr_Rolki_Wlot_1 : BOOL ;
  H1_Doj_Rolki_Wlot_1 : BOOL ;
  H2_Doj_Rolki_Wlot_1 : BOOL ;
  Filtr_Rolki_Wlot_2 : BOOL ;
  H1_Doj_Rolki_Wlot_2 : BOOL ;
  H2_Doj_Rolki_Wlot_2 : BOOL ;
  Pobranie_Wlot_1 : BOOL ;
  Pobranie_Wlot_2 : BOOL ;
  Paleta_Na_Obrotnicy : BOOL ;
  Oddanie_Palety : BOOL ;
  Help_Zez_Wlot_1 : BOOL ;
  Help_Zez_Wlot_2 : BOOL ;
  Obr_Na_Etykieciarke : BOOL ;
  Poz_Etykieciarka : BOOL ;
  Help_Silownik_Etyk : BOOL ;
  Oczekiwanie_Na_Obraz : BOOL ;
  Help_ety_przykl : BOOL ;
  Zbocze_przecisku_drukuj : BOOL ;
  Sprawdzenie_Etyk : BOOL ;
  Zbocze_1 : BOOL ;
  Zbocze_2 : BOOL ;
  Zbocze_3 : BOOL ;
  Zbocze_4 : BOOL ;
  H1 : BOOL ;
  H2 : BOOL ;
  H3 : BOOL ;
  H4 : BOOL ;
  H5 : BOOL ;
  H6 : BOOL ;
  H7 : BOOL ;
END_VAR
VAR_TEMP
  Temp_Help_1 : BOOL ;
  Temp_Help_2 : BOOL ;
  Czas_zadany : TIME ;
  Czas_aktualny : TIME ;
END_VAR
BEGIN
NETWORK
TITLE =
//                   
//Wlot 1                               Wylot
//()()()()|()()()()|  ()()()  |()()()()|()()()()
//()()()()|()()()()| ()()()() |()()()()|()()()()
//()()()()|()()()()| ()()()() |()()()()|()()()()
//()()()()|()()()()| ()()()() |()()()()|()()()()
//()()()()|()()()()|  ()()()  |()()()()|()()()()
//
//                  |()()()()|
//                  |()()()()|
//                  |()()()()| 
//                  |()()()()|
//                    Wlot_2
//         
//          pobierz --> zabierz   |     pobierz --> zabierz   
//     zez_od_nast <-- zez_do_pop | zez_od_nast <-- zez_od_pop
//                                  
//-Uklad dzielony jest na realizowane funkcje
//
//         
//                  
//
// ten network celowo jest pusty
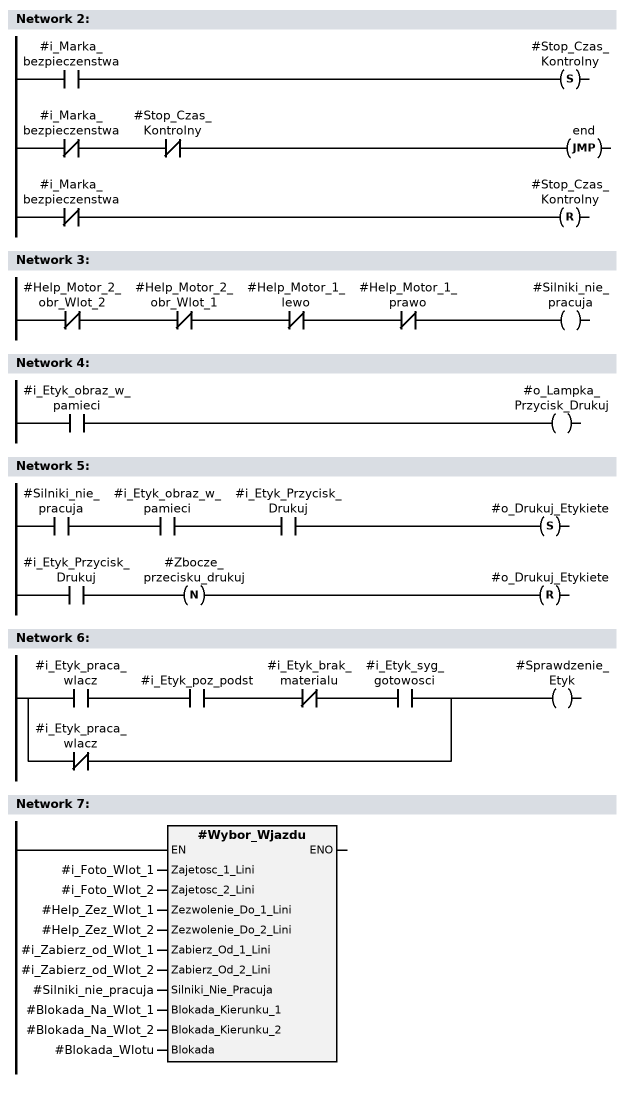
NETWORK
TITLE =
//Zatrzymanie uplywajacego czasu gdy brak bezpieczenstwa
//Skocz jezeli brak marki bezpieczenstwa
      A     #i_Marka_bezpieczenstwa;
      S     #Stop_Czas_Kontrolny;
      AN    #i_Marka_bezpieczenstwa;
      AN    #Stop_Czas_Kontrolny;
      JC    end;
      AN    #i_Marka_bezpieczenstwa;
      R     #Stop_Czas_Kontrolny;
NETWORK
TITLE =
//Sprawdzenie czy silniki nie pracuja
      AN    #Help_Motor_2_obr_Wlot_2;
      AN    #Help_Motor_2_obr_Wlot_1;
      AN    #Help_Motor_1_lewo;
      AN    #Help_Motor_1_prawo;
      =     #Silniki_nie_pracuja;
NETWORK
TITLE =
      A     #i_Etyk_obraz_w_pamieci;
      =     #o_Lampka_Przycisk_Drukuj;
NETWORK
TITLE =
//Drukowanie samej etykiety
      A     #Silniki_nie_pracuja;
      A     #i_Etyk_obraz_w_pamieci;
      A     #i_Etyk_Przycisk_Drukuj;
      S     #o_Drukuj_Etykiete;
      A     #i_Etyk_Przycisk_Drukuj;
      FN    #Zbocze_przecisku_drukuj;
      R     #o_Drukuj_Etykiete;
      NOP   0;
NETWORK
TITLE =
//Sprawdzenie etykietownicy zanim pobrana paleta
//Warunki pobrania palety gdy praca z etykietami
      A     #i_Etyk_praca_wlacz;
      A     #i_Etyk_poz_podst;
      AN    #i_Etyk_brak_materialu;	// gdy brak materialu
      A     #i_Etyk_syg_gotowosci;
      ON    #i_Etyk_praca_wlacz;
      =     #Sprawdzenie_Etyk;
NETWORK
TITLE =
//Wybranie wjazdu
      CALL  #Wybor_Wjazdu (
           Zajetosc_1_Lini          := #i_Foto_Wlot_1,
           Zajetosc_2_Lini          := #i_Foto_Wlot_2,
           Zezwolenie_Do_1_Lini     := #Help_Zez_Wlot_1,
           Zezwolenie_Do_2_Lini     := #Help_Zez_Wlot_2,
           Zabierz_Od_1_Lini        := #i_Zabierz_od_Wlot_1,
           Zabierz_Od_2_Lini        := #i_Zabierz_od_Wlot_2,
           Silniki_Nie_Pracuja      := #Silniki_nie_pracuja,
           Blokada_Kierunku_1       := #Blokada_Na_Wlot_1,
           Blokada_Kierunku_2       := #Blokada_Na_Wlot_2,
           Blokada                  := #Blokada_Wlotu);
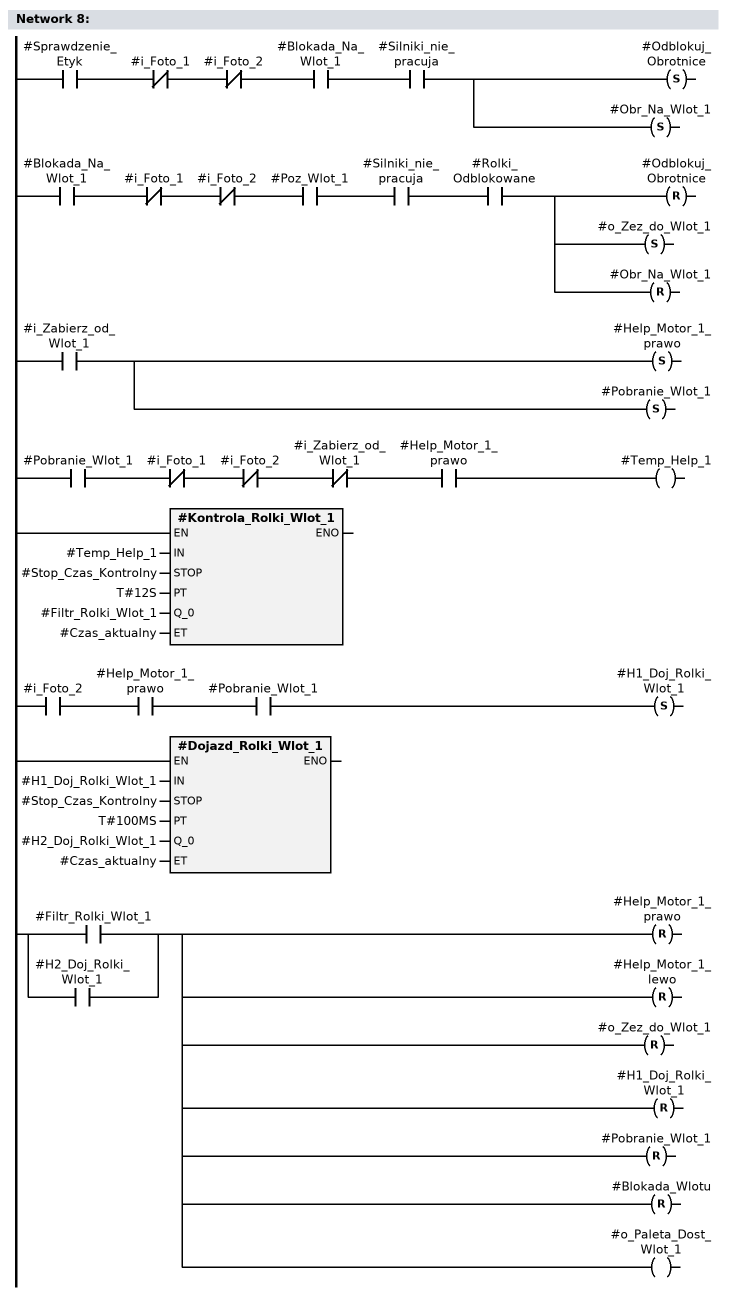
NETWORK
TITLE =
//Pobranie palety z Wlotu nr 1
//Obrot obrotnicy w kierunku wlotu nr 1
      A     #Sprawdzenie_Etyk;
      AN    #i_Foto_1;
      AN    #i_Foto_2;
      A     #Blokada_Na_Wlot_1;
      A     #Silniki_nie_pracuja;
      S     #Odblokuj_Obrotnice;
      S     #Obr_Na_Wlot_1;
//Zezwolenie na wjazd z wlotu 1
      A     #Blokada_Na_Wlot_1;
      AN    #i_Foto_1;
      AN    #i_Foto_2;
      A     #Poz_Wlot_1;
      A     #Silniki_nie_pracuja;
      A     #Rolki_Odblokowane;
      R     #Odblokuj_Obrotnice;
      S     #o_Zez_do_Wlot_1;
      R     #Obr_Na_Wlot_1;
//Gdy syganl zabierz to uruchom tasme
      A     #i_Zabierz_od_Wlot_1;
      S     #Help_Motor_1_prawo;
      S     #Pobranie_Wlot_1;
//Warunek gdy pobranie z poprzedniej i miejsce foto srodek
//jest zajete
      A     #Pobranie_Wlot_1;
      AN    #i_Foto_1;
      AN    #i_Foto_2;
      AN    #i_Zabierz_od_Wlot_1;
      A     #Help_Motor_1_prawo;
      =     #Temp_Help_1;
      CALL  #Kontrola_Rolki_Wlot_1 (
           IN                       := #Temp_Help_1,
           STOP                     := #Stop_Czas_Kontrolny,
           PT                       := T#12S,
           Q_0                      := #Filtr_Rolki_Wlot_1,
           ET                       := #Czas_aktualny);
      A     #i_Foto_2;
      A     #Help_Motor_1_prawo;
      A     #Pobranie_Wlot_1;
      S     #H1_Doj_Rolki_Wlot_1;
      CALL  #Dojazd_Rolki_Wlot_1 (
           IN                       := #H1_Doj_Rolki_Wlot_1,
           STOP                     := #Stop_Czas_Kontrolny,
           PT                       := T#100MS,
           Q_0                      := #H2_Doj_Rolki_Wlot_1,
           ET                       := #Czas_aktualny);
//Koniec pobierania palety z wlotu 1
      A     #Filtr_Rolki_Wlot_1;
      O;
      A     #H2_Doj_Rolki_Wlot_1;
      R     #Help_Motor_1_prawo;
      R     #Help_Motor_1_lewo;
      R     #o_Zez_do_Wlot_1;
      R     #H1_Doj_Rolki_Wlot_1;
      R     #Pobranie_Wlot_1;
      R     #Blokada_Wlotu;
      =     #o_Paleta_Dost_Wlot_1;
//-----------------------------------------------------
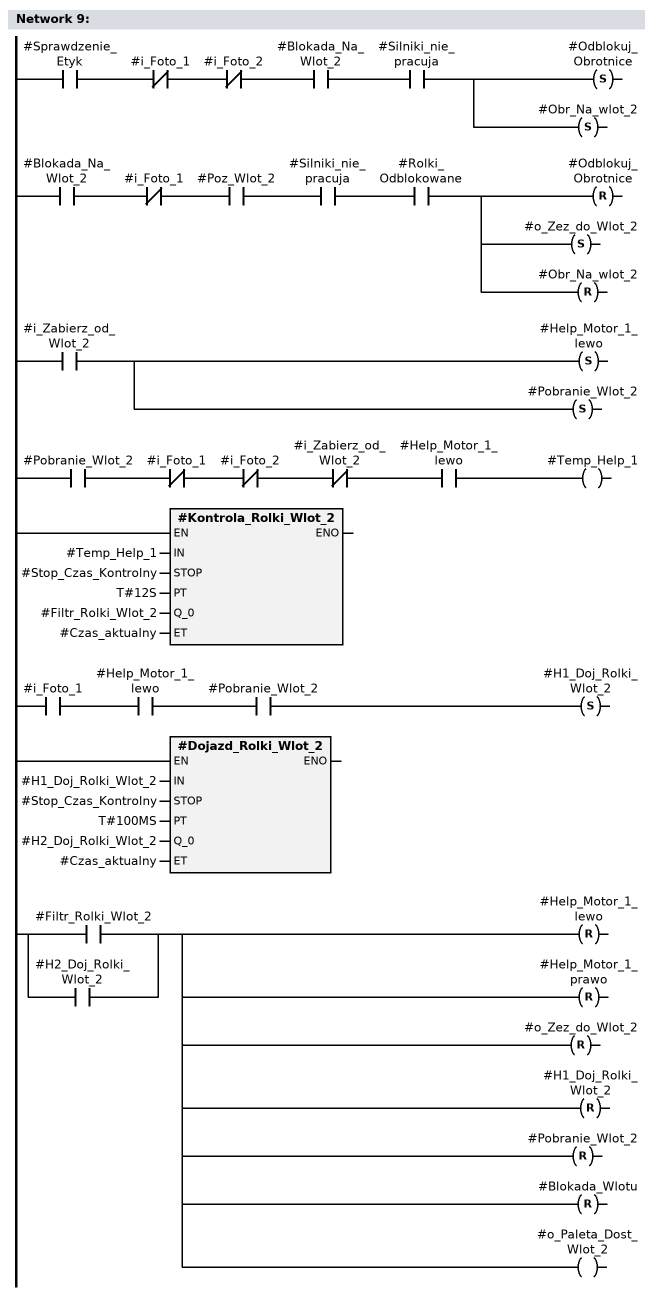
NETWORK
TITLE =
////Pobieranie Palety Wlot 2
//Obrot obrotnicy w kierunku wlotu nr 2
      A     #Sprawdzenie_Etyk;
      AN    #i_Foto_1;
      AN    #i_Foto_2;
      A     #Blokada_Na_Wlot_2;
      A     #Silniki_nie_pracuja;
      S     #Odblokuj_Obrotnice;
      S     #Obr_Na_wlot_2;
//Zezwolenie na wjazd z wlotu 2
      A     #Blokada_Na_Wlot_2;
      AN    #i_Foto_1;
      A     #Poz_Wlot_2;
      A     #Silniki_nie_pracuja;
      A     #Rolki_Odblokowane;
      R     #Odblokuj_Obrotnice;
      S     #o_Zez_do_Wlot_2;
      R     #Obr_Na_wlot_2;
//Gdy syganl zabierz to uruchom tasme
      A     #i_Zabierz_od_Wlot_2;
      S     #Help_Motor_1_lewo;
      S     #Pobranie_Wlot_2;
//Warunek gdy pobranie z poprzedniej i miejsce foto srodek
//jest zajete
      A     #Pobranie_Wlot_2;
      AN    #i_Foto_1;
      AN    #i_Foto_2;
      AN    #i_Zabierz_od_Wlot_2;
      A     #Help_Motor_1_lewo;
      =     #Temp_Help_1;
      CALL  #Kontrola_Rolki_Wlot_2 (
           IN                       := #Temp_Help_1,
           STOP                     := #Stop_Czas_Kontrolny,
           PT                       := T#12S,
           Q_0                      := #Filtr_Rolki_Wlot_2,
           ET                       := #Czas_aktualny);
      A     #i_Foto_1;
      A     #Help_Motor_1_lewo;
      A     #Pobranie_Wlot_2;
      S     #H1_Doj_Rolki_Wlot_2;
      CALL  #Dojazd_Rolki_Wlot_2 (
           IN                       := #H1_Doj_Rolki_Wlot_2,
           STOP                     := #Stop_Czas_Kontrolny,
           PT                       := T#100MS,
           Q_0                      := #H2_Doj_Rolki_Wlot_2,
           ET                       := #Czas_aktualny);
//Koniec pobierania palety z wlotu 2
      A     #Filtr_Rolki_Wlot_2;
      O;
      A     #H2_Doj_Rolki_Wlot_2;
      R     #Help_Motor_1_lewo;
      R     #Help_Motor_1_prawo;
      R     #o_Zez_do_Wlot_2;
      R     #H1_Doj_Rolki_Wlot_2;
      R     #Pobranie_Wlot_2;
      R     #Blokada_Wlotu;
      =     #o_Paleta_Dost_Wlot_2;
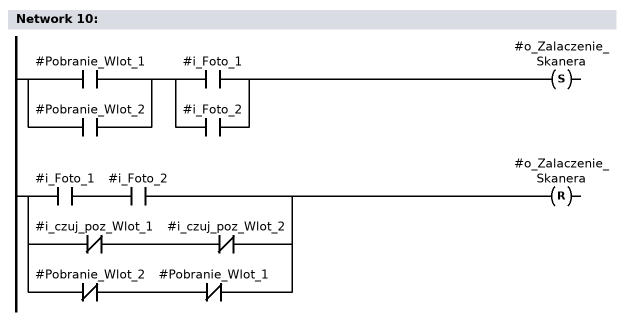
NETWORK
TITLE =
//Zalczenie skanera etykiet
      A(;
      O     #Pobranie_Wlot_1;
      O     #Pobranie_Wlot_2;
      );
      A(;
      O     #i_Foto_1;
      O     #i_Foto_2;
      );
      S     #o_Zalaczenie_Skanera;
      A(;
      A     #i_Foto_1;
      A     #i_Foto_2;
      O;
      AN    #i_czuj_poz_Wlot_1;
      AN    #i_czuj_poz_Wlot_2;
      O;
      AN    #Pobranie_Wlot_2;
      AN    #Pobranie_Wlot_1;
      );
      R     #o_Zalaczenie_Skanera;
      NOP   0;
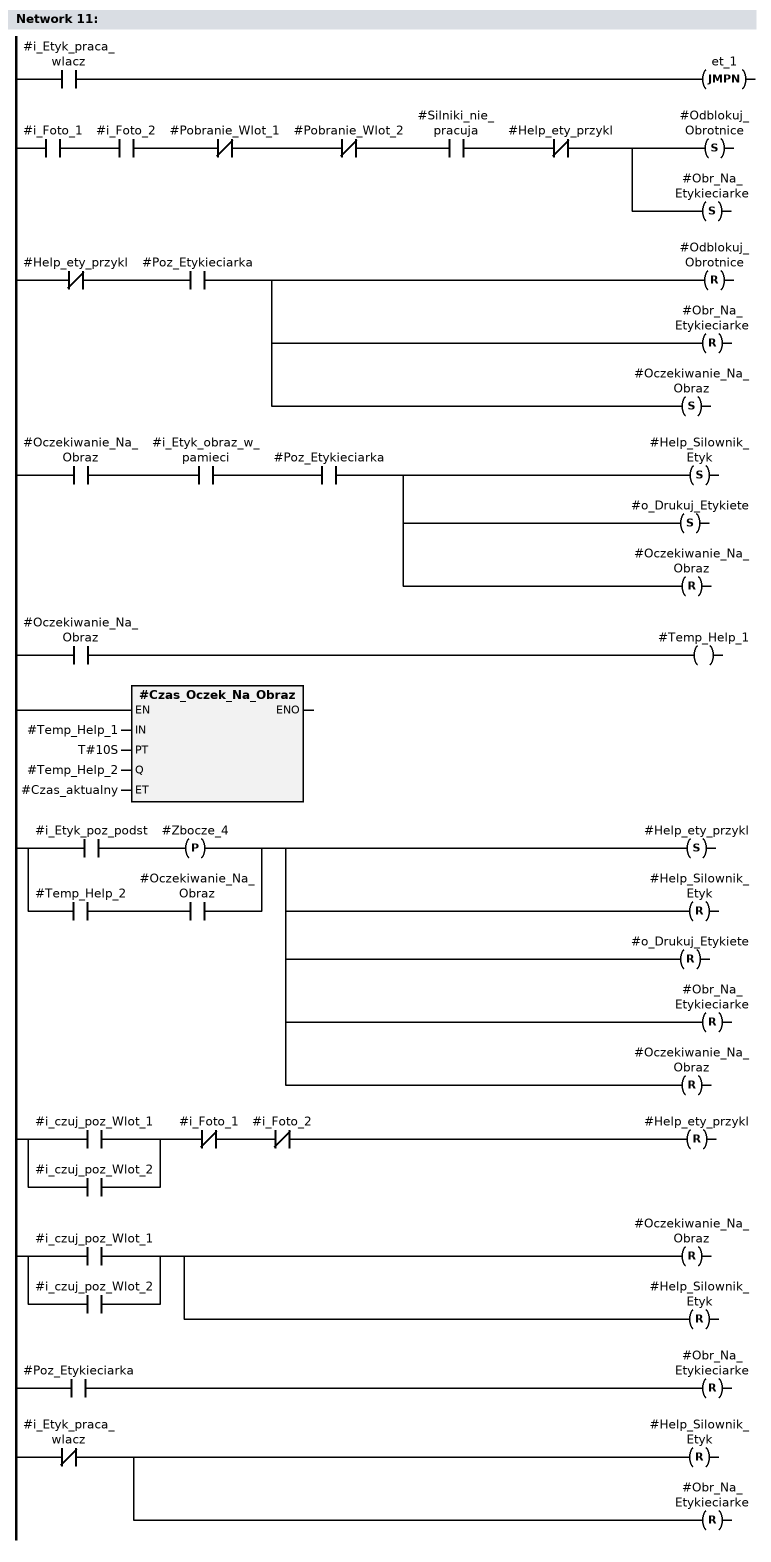
NETWORK
TITLE =
//Dojazd palety na etykieciarke
//Praca z etykietowaniem
      A     #i_Etyk_praca_wlacz;
      JCN   et_1;
// Obrot palety na maszyne etykietujaca
      A     #i_Foto_1;
      A     #i_Foto_2;
      AN    #Pobranie_Wlot_1;
      AN    #Pobranie_Wlot_2;
      A     #Silniki_nie_pracuja;
      AN    #Help_ety_przykl;
      S     #Odblokuj_Obrotnice;
      S     #Obr_Na_Etykieciarke;
//Oczekiwanie na
      AN    #Help_ety_przykl;
      A     #Poz_Etykieciarka;
      R     #Odblokuj_Obrotnice;
      R     #Obr_Na_Etykieciarke;
      S     #Oczekiwanie_Na_Obraz;
//Czas wstrzymania az obraz dotrze do etykieciarki
      A     #Oczekiwanie_Na_Obraz;
      A     #i_Etyk_obraz_w_pamieci;
      A     #Poz_Etykieciarka;	//dopisano 14.05.2014
      S     #Help_Silownik_Etyk;
      S     #o_Drukuj_Etykiete;
      R     #Oczekiwanie_Na_Obraz;
//Czas kontrolny oczekiwania na obraz
      A     #Oczekiwanie_Na_Obraz;
      =     #Temp_Help_1;
      CALL  #Czas_Oczek_Na_Obraz (
           IN                       := #Temp_Help_1,
           PT                       := T#10S,
           Q                        := #Temp_Help_2,
           ET                       := #Czas_aktualny);
//zakonczenie przyklejania etykiety
      A     #i_Etyk_poz_podst;
      FP    #Zbocze_4;
      O;
      A     #Temp_Help_2;
      A     #Oczekiwanie_Na_Obraz;
      S     #Help_ety_przykl;
      R     #Help_Silownik_Etyk;
      R     #o_Drukuj_Etykiete;
      R     #Obr_Na_Etykieciarke;
      R     #Oczekiwanie_Na_Obraz;	//dopisano 14.05.2014
//Warunkowy reset bitu przyklejania etykiety  
et_1: NOP   0;
      O     #i_czuj_poz_Wlot_1;
      O     #i_czuj_poz_Wlot_2;
      AN    #i_Foto_1;
      AN    #i_Foto_2;
      R     #Help_ety_przykl;
      O     #i_czuj_poz_Wlot_1;
      O     #i_czuj_poz_Wlot_2;
      R     #Oczekiwanie_Na_Obraz;
      R     #Help_Silownik_Etyk;
      A     #Poz_Etykieciarka;
      R     #Obr_Na_Etykieciarke;
      AN    #i_Etyk_praca_wlacz;
      R     #Help_Silownik_Etyk;
      R     #Obr_Na_Etykieciarke;
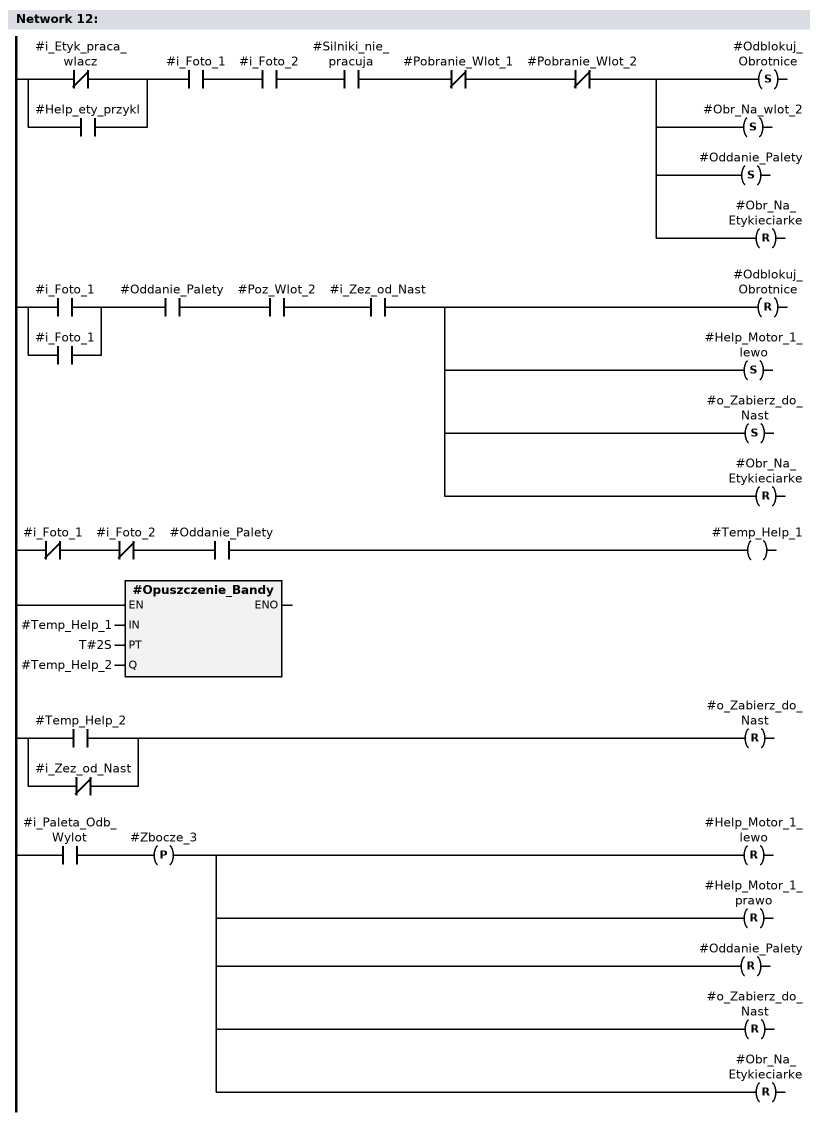
NETWORK
TITLE =
//Wyjazd palety z bandy obrotowej
//Jazda w kierunku wylotu
      ON    #i_Etyk_praca_wlacz;
      O     #Help_ety_przykl;
      A(;
      A     #i_Foto_1;
      A     #i_Foto_2;
      A     #Silniki_nie_pracuja;
      AN    #Pobranie_Wlot_1;
      AN    #Pobranie_Wlot_2;
      );
      S     #Odblokuj_Obrotnice;
      S     #Obr_Na_wlot_2;
      S     #Oddanie_Palety;
      R     #Obr_Na_Etykieciarke;
//Oczekiwanie na zezwolenie
      O     #i_Foto_1;
      O     #i_Foto_1;
      A     #Oddanie_Palety;
      A     #Poz_Wlot_2;
      A     #i_Zez_od_Nast;
      R     #Odblokuj_Obrotnice;
      S     #Help_Motor_1_lewo;
      S     #o_Zabierz_do_Nast;
      R     #Obr_Na_Etykieciarke;
//reset sygnalu zabierz
      AN    #i_Foto_1;
      AN    #i_Foto_2;
      A     #Oddanie_Palety;
      =     #Temp_Help_1;
      CALL  #Opuszczenie_Bandy (
           IN                       := #Temp_Help_1,
           PT                       := T#2S,
           Q                        := #Temp_Help_2);
      A     #Temp_Help_2;
      O;
      AN    #i_Zez_od_Nast;
      R     #o_Zabierz_do_Nast;
      A     #i_Paleta_Odb_Wylot;
//Otrzymanie sygalu zwrotnego o odbiorze palety
      FP    #Zbocze_3;
      R     #Help_Motor_1_lewo;
      R     #Help_Motor_1_prawo;
      R     #Oddanie_Palety;
      R     #o_Zabierz_do_Nast;
      R     #Obr_Na_Etykieciarke;
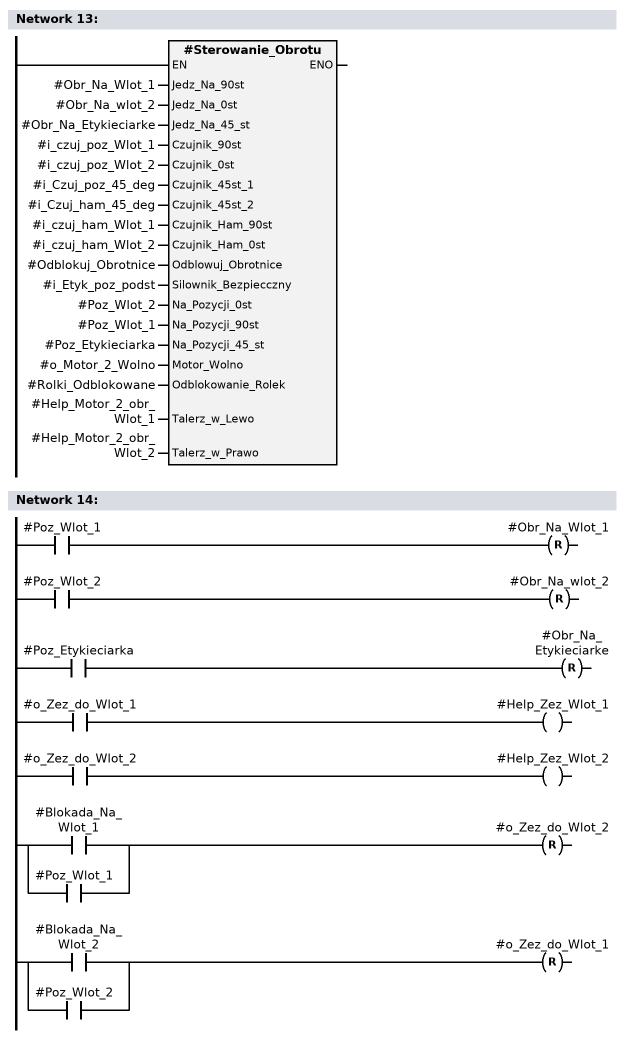
NETWORK
TITLE =
//Obrot na pozycje 
      CALL  #Sterowanie_Obrotu (
           Jedz_Na_90st             := #Obr_Na_Wlot_1,
           Jedz_Na_0st              := #Obr_Na_wlot_2,
           Jedz_Na_45_st            := #Obr_Na_Etykieciarke,
           Czujnik_90st             := #i_czuj_poz_Wlot_1,
           Czujnik_0st              := #i_czuj_poz_Wlot_2,
           Czujnik_45st_1           := #i_Czuj_poz_45_deg,
           Czujnik_45st_2           := #i_Czuj_ham_45_deg,
           Czujnik_Ham_90st         := #i_czuj_ham_Wlot_1,
           Czujnik_Ham_0st          := #i_czuj_ham_Wlot_2,
           Odblowuj_Obrotnice       := #Odblokuj_Obrotnice,
           Silownik_Bezpiecczny     := #i_Etyk_poz_podst,
           Na_Pozycji_0st           := #Poz_Wlot_2,
           Na_Pozycji_90st          := #Poz_Wlot_1,
           Na_Pozycji_45_st         := #Poz_Etykieciarka,
           Motor_Wolno              := #o_Motor_2_Wolno,
           Odblokowanie_Rolek       := #Rolki_Odblokowane,
           Talerz_w_Lewo            := #Help_Motor_2_obr_Wlot_1,
           Talerz_w_Prawo           := #Help_Motor_2_obr_Wlot_2);
NETWORK
TITLE =
//Warunki skrajne
      A     #Poz_Wlot_1;
      R     #Obr_Na_Wlot_1;
      A     #Poz_Wlot_2;
      R     #Obr_Na_wlot_2;
      A     #Poz_Etykieciarka;
      R     #Obr_Na_Etykieciarke;
      A     #o_Zez_do_Wlot_1;
      =     #Help_Zez_Wlot_1;
      A     #o_Zez_do_Wlot_2;
      =     #Help_Zez_Wlot_2;
      O     #Blokada_Na_Wlot_1;
      O     #Poz_Wlot_1;
      R     #o_Zez_do_Wlot_2;
      O     #Blokada_Na_Wlot_2;
      O     #Poz_Wlot_2;
      R     #o_Zez_do_Wlot_1;
NETWORK
TITLE =
//Warunki skrajne
end:  NOP   0;
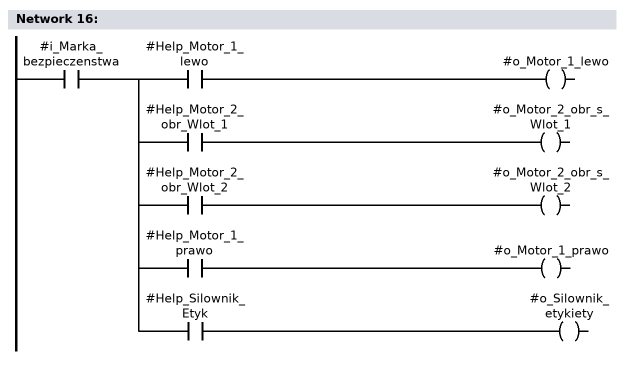
NETWORK
TITLE =
      A     #i_Marka_bezpieczenstwa;
      =     L 10.0;
      A     L 10.0;
      A     #Help_Motor_1_lewo;
      =     #o_Motor_1_lewo;
      A     L 10.0;
      A     #Help_Motor_2_obr_Wlot_1;
      =     #o_Motor_2_obr_s_Wlot_1;
      A     L 10.0;
      A     #Help_Motor_2_obr_Wlot_2;
      =     #o_Motor_2_obr_s_Wlot_2;
      A     L 10.0;
      A     #Help_Motor_1_prawo;
      =     #o_Motor_1_prawo;
      A     L 10.0;
      A     #Help_Silownik_Etyk;
      =     #o_Silownik_etykiety;
NETWORK
TITLE =
END_FUNCTION_BLOCK

FUNCTION_BLOCK "Banda_Poj_+Tryb_Reczny"	// FB 33
//Funkcja realizujaca koncepcje bandy pojedycznej, ktora uwzglednia rowniez tryb 
//reczny. W celu lepszego sterowania trybem recznym nalezy do³o¿yæ:
//-fotokomorki na tyle bandy.
//-fotokomorka na tyle okresla rowniez zajetosc
//-jazda do tylu bandy mozliwa
//-jazda do przodu poza fotokomorke mozliwa gdy nastepna w ruchu i wolna.
//-do³o¿enie okresnia trybu reczny/auto gdzie auto to 1 
//
AUTHOR : Kng
FAMILY : Bandy
NAME : B_dual
VERSION : 0.0
VAR_INPUT
  i_Marka_Bezpieczenstwa : BOOL ;
  i_Rezerwa_1 : BOOL ;	//Zamrozenie stanu pracy
  i_Auto_Reczny : BOOL ;	//1-auto,0-reczny
  i_Foto_Przod : BOOL ;	//Foto na koncu tasmy
  i_Foto_Tyl : BOOL ;	//Foto zapobiegajace wyjechaniu palety do tylu
  i_Zez_Od_Nast : BOOL ;
  i_Paleta_Dost_Od_Nast : BOOL ;
  i_Zez_Reczny_Od_Nast : BOOL ;
  i_Zabierz_Od_Pop : BOOL ;
  i_Zez_Reczny_Od_Pop : BOOL ;
  i_PB_Jazda_Tyl : BOOL ;
  i_PB_Jazda_Przod : BOOL ;
  Czas_Kontroli_Przejazdu : TIME ;
END_VAR
VAR_OUTPUT
  o_Zabierz_Do_Nast : BOOL ;	//Rozkaz pobrania do nast bandy
  o_Zez_Do_Pop : BOOL ;
  o_Paleta_Dost_Do_Pop : BOOL ;
  o_Motor_Lewo : BOOL ;
  o_Motor_Prawo : BOOL ;
  o_Zez_Reczny_Do_Nast : BOOL ;
  o_Zez_Reczny_Do_Pop : BOOL ;
  o_Zajetosc_Nieb : BOOL ;	//Dla bezpieczenstwa transportu
END_VAR
VAR
  Czas_kontrolny : FB 21;
  Help_A_Motor_Lewo : BOOL ;
  S_Help_Zab_Od_Pop : BOOL ;
  Stop_Czas_Kontrolny : BOOL ;
  Zbocze_1 : BOOL ;
  Zbocze_2 : BOOL ;
  Blokada_Wjazdu : BOOL ;
  Help_H_Motor_Prawo : BOOL ;
  Help_H_Motor_Lewo : BOOL ;
  Toggle : BOOL ;	//bit przemienny dla auto i hand
  Help_8 : BOOL ;
  Help_9 : BOOL ;
END_VAR
VAR_TEMP
  Temp_Help_1 : BOOL ;
  Temp_Help_2 : BOOL ;
  Czas_zadany : TIME ;
  Czas_aktualny : TIME ;
END_VAR
BEGIN
NETWORK
TITLE =
//
// B1        B2         foto_1    foto_2         B5        B6
//(\\\\\\\\\\\\\\\\\\)  (\\\\\\\\\\\\\\\\\\)  (\\\\\\\\\\\\\\\\\\)
//                  M1                    M2                     M3
//         
//        zabierz <-- pobierz      |  zabierz    <--  pobierz  
//     zez_do_pop --> zez_od_nast  |  zez_od_pop -->  zez_od_nast
//                                  
//-Uklad dzielony jest na realizowane funkcje
//
//         <----------------------------------------- kierunek
//                  
//
// ten network celowo jest pusty
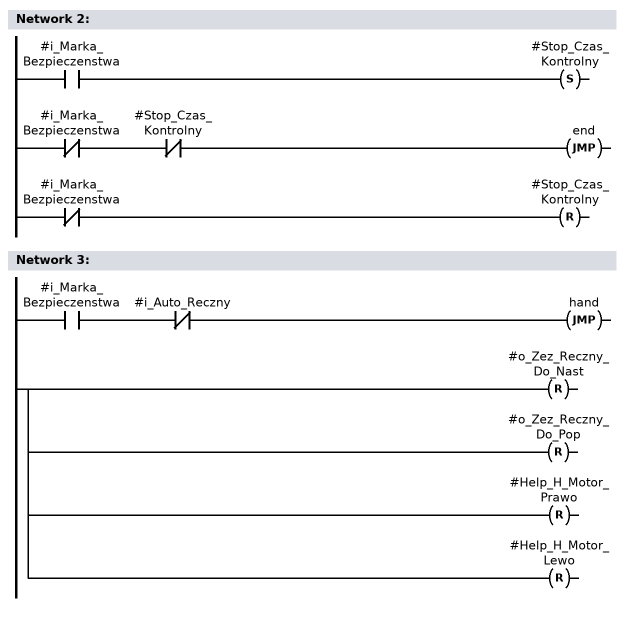
NETWORK
TITLE =
//Sprawdzenie stanu bezpieczenstwa lub freeze
//Skocz jezeli brak marki bezpieczenstwa
//Marka bezpieczenstwa ok gdy wysoki
      A     #i_Marka_Bezpieczenstwa;
      S     #Stop_Czas_Kontrolny;
      AN    #i_Marka_Bezpieczenstwa;
      AN    #Stop_Czas_Kontrolny;
      JC    end;
      AN    #i_Marka_Bezpieczenstwa;
      R     #Stop_Czas_Kontrolny;
NETWORK
TITLE =
//Wyznczenie zbocza pozytywnego i negatywnego
//skok do trybu recznego 
      A     #i_Marka_Bezpieczenstwa;
      AN    #i_Auto_Reczny;
      JC    hand;
//czyszczenie trybu recznego
      SET;
      R     #o_Zez_Reczny_Do_Nast;
      R     #o_Zez_Reczny_Do_Pop;
      R     #Help_H_Motor_Prawo;
      R     #Help_H_Motor_Lewo;
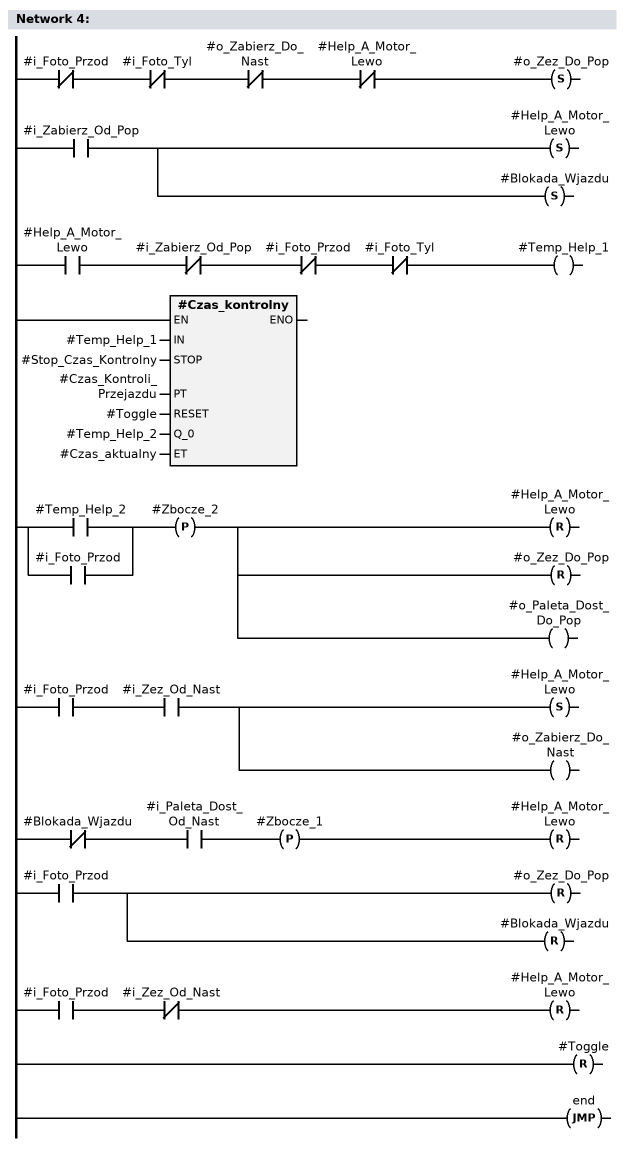
NETWORK
TITLE =
// Opis poszczegolnych krokow i skok do nich
// Tasma poprzednia pusta i bierzaca pusta
      AN    #i_Foto_Przod;
      AN    #i_Foto_Tyl;	//dodano bo hand
      AN    #o_Zabierz_Do_Nast;
      AN    #Help_A_Motor_Lewo;
      S     #o_Zez_Do_Pop;
      A     #i_Zabierz_Od_Pop;
      S     #Help_A_Motor_Lewo;
      S     #Blokada_Wjazdu;
//Warunek gdy pobranie z poprzedniej i miejsce foto srodek
//jest zajete
      A     #Help_A_Motor_Lewo;
      AN    #i_Zabierz_Od_Pop;
      AN    #i_Foto_Przod;
      AN    #i_Foto_Tyl;	//dodano bo hand
      =     #Temp_Help_1;
      CALL  #Czas_kontrolny (
           IN                       := #Temp_Help_1,
           STOP                     := #Stop_Czas_Kontrolny,
           PT                       := #Czas_Kontroli_Przejazdu,
           RESET                    := #Toggle,
           Q_0                      := #Temp_Help_2,
           ET                       := #Czas_aktualny);
//Paleta dostarczona
      A     #Temp_Help_2;
      O;
      A     #i_Foto_Przod;
      FP    #Zbocze_2;
      R     #Help_A_Motor_Lewo;
      R     #o_Zez_Do_Pop;
      =     #o_Paleta_Dost_Do_Pop;
//jest zezwolenie od nastepnej
      A     #i_Foto_Przod;
      A     #i_Zez_Od_Nast;
      S     #Help_A_Motor_Lewo;
      =     #o_Zabierz_Do_Nast;
//Potwierdzenie otrzymania palety
      AN    #Blokada_Wjazdu;
      A     #i_Paleta_Dost_Od_Nast;
      FP    #Zbocze_1;
      R     #Help_A_Motor_Lewo;
//Gdy zajete Foto_1 brak zezwolenia do poprzedniej
      A     #i_Foto_Przod;
      R     #o_Zez_Do_Pop;
      R     #Blokada_Wjazdu;
//warunkowe zakonczenie pracy silnika gdy brak zezwolenia
//z nastepnej
      A     #i_Foto_Przod;
      AN    #i_Zez_Od_Nast;
      R     #Help_A_Motor_Lewo;
//wylacz toggle
      SET;
      R     #Toggle;
//skocz do koniec
      JU    end;
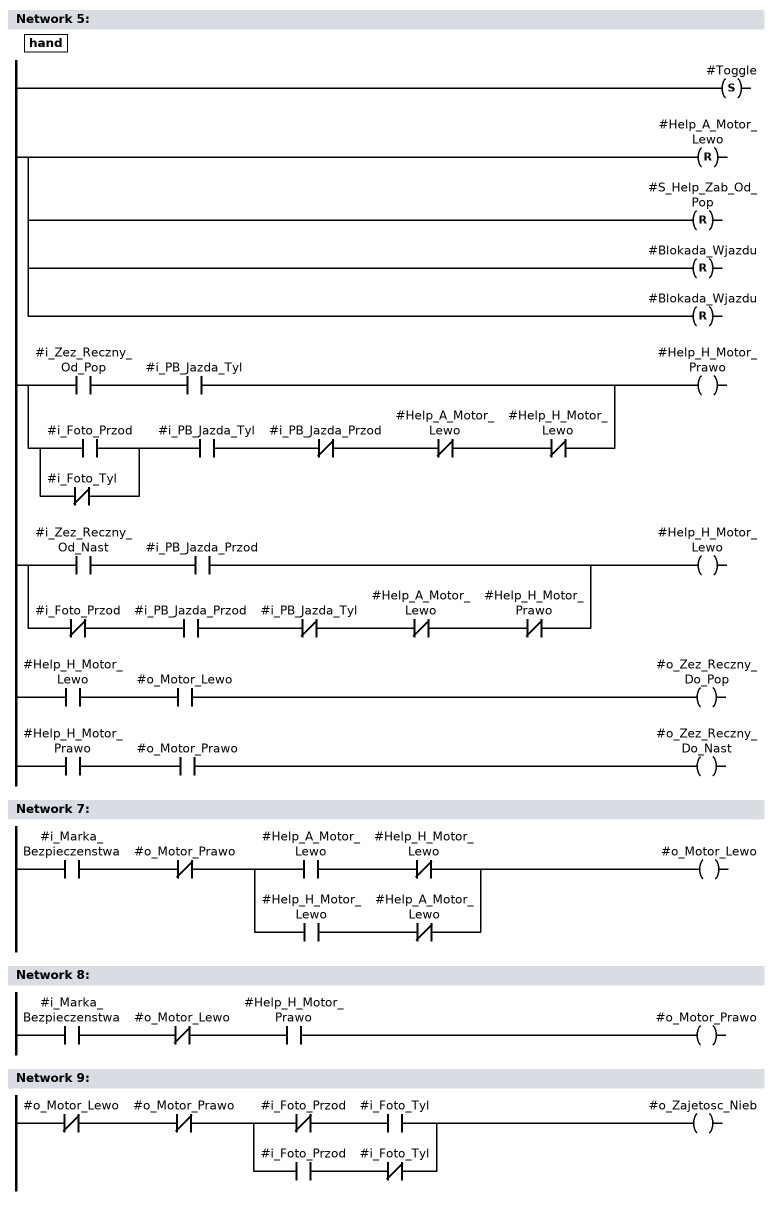
NETWORK
TITLE =
//Tryb reczny
//
hand: NOP   0;
//wlacz toggle
      SET;
      S     #Toggle;
//czyszczenie bitow z automatyki
      SET;
      R     #Help_A_Motor_Lewo;
      R     #S_Help_Zab_Od_Pop;
      R     #Blokada_Wjazdu;
      R     #Blokada_Wjazdu;
//ustawienie przyciskow
//jazda do tylu przycisk tyl
      A     #i_Zez_Reczny_Od_Pop;
      A     #i_PB_Jazda_Tyl;
      O;
      A(;
      O     #i_Foto_Przod;
      ON    #i_Foto_Tyl;
      );
      A(;
      A     #i_PB_Jazda_Tyl;
      AN    #i_PB_Jazda_Przod;
      AN    #Help_A_Motor_Lewo;
      AN    #Help_H_Motor_Lewo;
      );
      =     #Help_H_Motor_Prawo;
//jazda do przodu
      A     #i_Zez_Reczny_Od_Nast;
      A     #i_PB_Jazda_Przod;
      O;
      AN    #i_Foto_Przod;
      A(;
      A     #i_PB_Jazda_Przod;
      AN    #i_PB_Jazda_Tyl;
      AN    #Help_A_Motor_Lewo;
      AN    #Help_H_Motor_Prawo;
      );
      =     #Help_H_Motor_Lewo;
//wystawienie zezwolen do innych band wspolpracujacych recznie
//zezwolenie do tylu 
//zezwolenie do poprzedniej
      A     #Help_H_Motor_Lewo;
      A     #o_Motor_Lewo;
      =     #o_Zez_Reczny_Do_Pop;
//zezwolenie do nastepnej
      A     #Help_H_Motor_Prawo;
      A     #o_Motor_Prawo;
      =     #o_Zez_Reczny_Do_Nast;
NETWORK
TITLE =
//Przypisanie wyjsc
//Koniec skoku
end:  NOP   0;
NETWORK
TITLE =
////jazda automatyka reczny przod
      A     #i_Marka_Bezpieczenstwa;
      AN    #o_Motor_Prawo;
      A(;
      A     #Help_A_Motor_Lewo;
      AN    #Help_H_Motor_Lewo;
      O;
      A     #Help_H_Motor_Lewo;
      AN    #Help_A_Motor_Lewo;
      );
      =     #o_Motor_Lewo;
NETWORK
TITLE =
////Jazda reczny tyl
      A     #i_Marka_Bezpieczenstwa;
      AN    #o_Motor_Lewo;
      A     #Help_H_Motor_Prawo;
      =     #o_Motor_Prawo;
NETWORK
TITLE =
//Zajetosc
      AN    #o_Motor_Lewo;
      AN    #o_Motor_Prawo;
      A(;
      AN    #i_Foto_Przod;
      A     #i_Foto_Tyl;
      O;
      A     #i_Foto_Przod;
      AN    #i_Foto_Tyl;
      );
      =     #o_Zajetosc_Nieb;
NETWORK
TITLE =
//Koniec
//koniec
      BEU;
END_FUNCTION_BLOCK

FUNCTION_BLOCK "Banda_Obr_Bind"	// FB 34
//Program odpowiadajacy za bindowanie produktu na obrotnicy
//
//
AUTHOR : Kng
FAMILY : Bandy
NAME : Band_obr
VERSION : 0.1
VAR_INPUT
  i_Marka_Bezpieczenstwa : BOOL ;
  i_Auto_Reczny : BOOL ;	//gdzie 1-Auto 0 Reczny
  i_Bindownica_Auto : BOOL ;	//Mro¿enie stanu pracy
  i_Foto_Tyl : BOOL ;	//foto poczatek
  i_Foto_Przod : BOOL ;	//foto koniec
  i_Zez_od_Nast : BOOL ;
  i_Zabierz_od_Pop : BOOL ;
  i_Paleta_Dost_Od_Nast : BOOL ;
  i_czuj_0_st_1 : BOOL ;	//0 stopni Wlot/Wylot
  i_czuj_0_st_2 : BOOL ;	//Hamowanie 0 stopni
  i_czuj_90_st_1 : BOOL ;	//Hamowanie 90 stopni
  i_czuj_90_st_2 : BOOL ;	//90 stopni
  i_Czuj_180_st_1 : BOOL ;	//Hamowanie 180 stopni
  i_Czuj_180_st_2 : BOOL ;	//180 stopni
  i_Czuj_270_st_1 : BOOL ;	//Hamowanie 270 stopni
  i_Czuj_270_st_2 : BOOL ;
  i_Bind_Obwod_Ok : BOOL ;	//270 stopni
  i_Bind_Poz_Podst : BOOL ;
  i_Bind_Syg_Got : BOOL ;
  i_Bind_Blad : BOOL ;
  i_Bind_Start_Kon : BOOL ;	//Bindownica start koniec wiazania
  i_PB_Obr_Prawo : BOOL ;
  i_PB_Obr_Lewo : BOOL ;
  i_Zawsze_True : BOOL ;	//Zawsze jeden do pomocy
  i_PB_Jazda_Przod : BOOL ;
  i_PB_Jazda_Tyl : BOOL ;
  i_PB_Cykl_Start : BOOL ;
  i_PB_Cykl_Stop : BOOL ;
  i_Zez_Reczny_Od_Pop : BOOL ;
  i_Zez_Reczny_Od_Nast : BOOL ;
  i_Reset_Krokow : BOOL ;
  i_Reset_Bledow : BOOL ;
  i_Rezerwa_1 : BOOL ;
  i_Rezerwa_2 : BOOL ;
  i_Rezerwa_3 : BOOL ;
  i_Rezerwa_4 : BOOL ;
END_VAR
VAR_OUTPUT
  o_Zez_do_Pop : BOOL ;
  o_Paleta_Dost_Do_Pop : BOOL ;
  o_Zabierz_do_Nast : BOOL ;
  o_Motor_1_lewo : BOOL ;
  o_Motor_1_prawo : BOOL ;
  o_Motor_1_Wolno : BOOL ;
  o_Motor_2_obr_s_Lewo : BOOL ;	//Motor obrotnicy,kierunek strona wejscia,szybko
  o_Motor_2_obr_s_Prawo : BOOL ;	//Motor obrotnicy,kierunek strona wyjscia,szybko
  o_Motor_2_Wolno : BOOL ;	//Motor obrotnicy,kierunek strona wejscia,wolno
  o_Bind_Zez_Na_Prace : BOOL ;
  o_Bind_Start_Wiazania : BOOL ;
  o_Bind_Blad_Ogolny : BOOL ;
  o_Zez_Reczny_do_Pop : BOOL ;
  o_Zez_Reczny_do_nast : BOOL ;
  o_Lampka_Bindowanie : BOOL ;
  o_Lampka_Przycisk_Reset : BOOL ;
  o_Blad_Cyklu : BOOL ;
  o_Blad_Ogolny : BOOL ;
  o_Cykl_Bindowania_Trwa : BOOL ;
  o_Rezerwa_2 : BOOL ;
  o_Rezerwa_3 : BOOL ;
END_VAR
VAR
  Sterowanie_Obrotu : FB 54;
  Pozycj_Obr : FB 55;
  Bindowanie : FB 35;
  Pozycjonowanie_Palety : FB 58;
  Kontrola_Rolki_Wlot : FB 20;
  Dojazd_Rolki_Wlot : FB 20;
  Opuszczenie_Bandy : FB 20;	//Czas kontrolny wjazdu palety
  Tim_Rezerwa_1 : FB 20;
  Tim_Rezerwa_2 : FB 20;
  Tim_Rezerwa_3 : SFB 4;	//Timer opozniajacy bindowanie
  Silniki_nie_pracuja : BOOL ;
  Help_A_Motor_1_lewo : BOOL ;
  Help_A_Motor_1_prawo : BOOL ;
  Help_A_Motor_1_wolno : BOOL ;
  Help_H_Motor_1_lewo : BOOL ;
  Help_H_Motor_1_prawo : BOOL ;
  Help_H_Motor_1_Wolno : BOOL ;
  Help_Motor_2_obr_lewo : BOOL ;
  Help_Motor_2_obr_prawo : BOOL ;
  Help_Motor_2_Wolno : BOOL ;
  Help_AP_Motor_1_Lewo : BOOL ;
  Help_AP_Motor_1_Prawo : BOOL ;
  Help_AP_Motor_1_Wolno : BOOL ;
  Pobranie_Wlot : BOOL ;
  Filtr_Rolki_Wlot : BOOL ;
  Stop_Czas_Kontrolny : BOOL ;
  H1_Doj_Rolki_Wlot : BOOL ;
  H2_Doj_Rolki_Wlot : BOOL ;
  Oddanie_Palety : BOOL ;
  Zbocze_1 : BOOL ;
  Toggle : BOOL ;	//Sygnal zamienny auto reczny
  Paleta_rowno_na_stan : BOOL ;
  Help_B_Zez_Na_Prace : BOOL ;
  Help_B_Start_Wiazan : BOOL ;
  Help_B_Blad_Ogolny : BOOL ;
  Help_Bin_Koniec_Cyklu : BOOL ;
  H_Start_Cyklu_Bind_Auto : BOOL ;
  H_Reset_Cyklu_Bind : BOOL ;
  H_Auto_Reczny : BOOL ;
  Auto_Reczny_W : BOOL ;
  Silnik_Rolek_Nie_Pracuje : BOOL ;
  Reset_Konca_Cyklu : BOOL ;
  Zbocze_2 : BOOL ;
  Help_PB_Start : BOOL ;
  H_Silnik_Rolek_Pracuje : BOOL ;
  H_Zez_do_Pop : BOOL ;
  H_Zabierz_do_Nast : BOOL ;
  H_Cykl_Bind_Trwa : BOOL ;
  Zbocze_3 : BOOL ;
  H_Blad_Cyklu : BOOL ;
  H_Marka_Bezp_Obr : BOOL ;
  H_Marka_Bezp_Poz : BOOL ;
  H_Auto_Reczny_Ster_Obr : BOOL ;
  H_Start_Cyklu_Bind_Recz : BOOL ;
  H_Reset_Srodka : BOOL ;	//Reset paleta na srodku
  H2_Start_Cyklu_Bind_Recz : BOOL ;
  H46 : BOOL ;
  H49 : BOOL ;
  H50 : BOOL ;
  Help_Cykl_Start_Reczny : BOOL ;
  H52 : BOOL ;
  H54 : BOOL ;
  H55 : BOOL ;
  H56 : BOOL ;
  H57 : BOOL ;
  H58 : INT ;
  H59 : BOOL ;
  H60 : BOOL ;	//Pozycja talerza osiagnieta
  H62 : BOOL ;
  H61 : INT ;
  H63 : BOOL ;
  H64 : BOOL ;
  H65 : BOOL ;
  H66 : BOOL ;
  H67 : BOOL ;
  H68 : BOOL ;
  H69 : BOOL ;
  H70 : BOOL ;
  H72 : BOOL ;
  H40 : BOOL ;
  H38 : BOOL ;
  H37 : BOOL ;
  H36 : BOOL ;
  H35 : BOOL ;
  H34 : BOOL ;
  H33 : BOOL ;
  H32 : BOOL ;
  H31 : BOOL ;
  H30 : BOOL ;
  H29 : BOOL ;
  H28 : BOOL ;	//Pozycjonowanie palety
  H27 : BOOL ;
  H26 : BOOL ;
END_VAR
VAR_TEMP
  Temp_Help_1 : BOOL ;
  Temp_Help_2 : BOOL ;
  Czas_zadany : TIME ;
  Czas_aktualny : TIME ;
  Czas_Kontroli_Przejazdu : TIME ;
  Czas_Monitora_Najazdu : TIME ;
  Czas_Opoznienia_Bind : TIME ;
END_VAR
BEGIN
NETWORK
TITLE =
//                   
//Wlot                                Wylot
//()()()()|()()()()|  ()()()  |()()()()|()()()()
//()()()()|()()()()| ()()()() |()()()()|()()()()
//()()()()|()()()()| ()()()() |()()()()|()()()()
//()()()()|()()()()| ()()()() |()()()()|()()()()
//()()()()|()()()()|  ()()()  |()()()()|()()()()
//
//      
//         
//          pobierz --> zabierz   |     pobierz --> zabierz   
//     zez_od_nast <-- zez_do_pop | zez_od_nast <-- zez_od_pop
//                                  
//-Uklad dzielony jest na realizowane funkcje
//
//         
//                  
//
// ten network celowo jest pusty
NETWORK
TITLE =
//Wyznczenie zbocza pozytywnego i negatywnego
//Skocz jezeli brak marki bezpieczenstwa
//Marka bezpieczenstwa ok gdy wysoki
//Freeze ok gdy niski
      A     #i_Marka_Bezpieczenstwa;
      S     #Stop_Czas_Kontrolny;
//skocz aby zrobic reset podczas stopu
      AN    #Stop_Czas_Kontrolny;
      A     #i_Reset_Krokow;
      JC    bind;
      AN    #i_Marka_Bezpieczenstwa;
      AN    #Stop_Czas_Kontrolny;
      JC    end;
      AN    #i_Marka_Bezpieczenstwa;
      R     #Stop_Czas_Kontrolny;
NETWORK
TITLE =
//Sprawdzenie czy rolki nie pracuja 
      AN    #Help_AP_Motor_1_Lewo;
      AN    #Help_AP_Motor_1_Prawo;
      AN    #Help_A_Motor_1_lewo;
      AN    #Help_A_Motor_1_prawo;
      AN    #Help_H_Motor_1_lewo;
      AN    #Help_H_Motor_1_prawo;
      =     #Silnik_Rolek_Nie_Pracuje;
      A     #Silnik_Rolek_Nie_Pracuje;
      NOT;
      =     #H_Silnik_Rolek_Pracuje;
NETWORK
TITLE =
//Silniki nie pracuja
//
      A     #Silnik_Rolek_Nie_Pracuje;
      AN    #Help_Motor_2_obr_lewo;
      AN    #Help_Motor_2_obr_prawo;
      =     #Silniki_nie_pracuja;
NETWORK
TITLE =
//Sprawdzenie czy paleta lezy na stanowisku
//sprawdzenie czy paleta lezy OK
      A     #i_Foto_Przod;
      A     #i_Foto_Tyl;
      =     #Paleta_rowno_na_stan;
NETWORK
TITLE =
//Skok do trybu recznego 
//skok do trybu recznego 
      A     #i_Marka_Bezpieczenstwa;
      AN    #i_Auto_Reczny;
      JC    hand;
//Powrot z trybu recznego do auto
      A     #Toggle;
      R     #Oddanie_Palety;
//czyszczenie trybu recznego
      SET;
      R     #o_Zez_Reczny_do_nast;
      R     #o_Zez_Reczny_do_Pop;
      R     #Help_H_Motor_1_prawo;
      R     #Help_H_Motor_1_lewo;
      R     #Auto_Reczny_W;
NETWORK
TITLE =
//Wjazd palety na stanowisko bindowania
// Opis poszczegolnych krokow i skok do nich
// Tasma poprzednia pusta i bierzaca pusta
      AN    #i_Foto_Przod;
      AN    #i_Foto_Tyl;
      AN    #H_Zabierz_do_Nast;
      A     #Silniki_nie_pracuja;
      A     #i_Bind_Poz_Podst;
      A     "Blok_Para".Poz_0_st;
      A     "Blok_Para".Odblokuj_Rolki;
      S     #H_Zez_do_Pop;
//gdy sygnal zabierzto blokada wjazdu
      A     #i_Zabierz_od_Pop;
      S     #Help_A_Motor_1_lewo;
      S     #Pobranie_Wlot;
//Czas kontrolny wjazdu na bande
      A     #Pobranie_Wlot;
      AN    #i_Foto_Przod;
      AN    #i_Foto_Tyl;
      AN    #i_Zabierz_od_Pop;
      A     #Help_A_Motor_1_lewo;
      =     #Temp_Help_1;
//Czas kontrolny dojazdu na stanowisko pracy
      CALL  #Kontrola_Rolki_Wlot (
           IN                       := #Temp_Help_1,
           STOP                     := #Stop_Czas_Kontrolny,
           PT                       := T#20S,
           Q_0                      := #Filtr_Rolki_Wlot,
           ET                       := #Czas_aktualny);
//Dojazd na pozycje na obrotnicy
      A     #i_Foto_Przod;
      A     #Help_A_Motor_1_lewo;
      A     #Pobranie_Wlot;
      S     #H1_Doj_Rolki_Wlot;
      S     #Help_A_Motor_1_wolno;
      CALL  #Dojazd_Rolki_Wlot (
           IN                       := #H1_Doj_Rolki_Wlot,
           STOP                     := #Stop_Czas_Kontrolny,
           PT                       := T#1S500MS,
           Q_0                      := #H2_Doj_Rolki_Wlot,
           ET                       := #Czas_aktualny);
//Koniec pobierania palety z wlotu 1
      A     #Filtr_Rolki_Wlot;
      O;
      A     #H2_Doj_Rolki_Wlot;
      R     #Help_A_Motor_1_lewo;
      R     #H_Zez_do_Pop;
      R     #H1_Doj_Rolki_Wlot;
      R     #Pobranie_Wlot;
      R     #Help_A_Motor_1_wolno;
      =     #o_Paleta_Dost_Do_Pop;
//-------------------------------------------------
NETWORK
TITLE = //wyjazd wtrybie auto
//Bindowanie
//rozpoczecie cyklu bindowania
      A     "Auto_Reczny";
      A     #Paleta_rowno_na_stan;
      A     #o_Paleta_Dost_Do_Pop;
      S     #H_Start_Cyklu_Bind_Auto;
//zakolnczenie cyku bindowania
      O     #Oddanie_Palety;
      ON    #i_Auto_Reczny;
      O     #H_Cykl_Bind_Trwa;
      O(;
      AN    #i_Foto_Przod;
      AN    #i_Foto_Tyl;
      );
      R     "Blok_Para".Trigger_Wyjazd;
      A     "Auto_Reczny";
      A(;
      O     #Help_Bin_Koniec_Cyklu;
      O     "Blok_Para".Trigger_Wyjazd;
      );
      S     #Oddanie_Palety;
NETWORK
TITLE =
//Wyjazd palety z bindowania
//jest zezwolenie od nastepnej
//Oczekiwanie na zezwolenie
      O     #i_Foto_Przod;
      O     #i_Foto_Tyl;
      A     #Oddanie_Palety;
      A     "Blok_Para".Odblokuj_Rolki;
      A     "Blok_Para".Poz_0_st;
      A     #i_Zez_od_Nast;
      S     #Help_A_Motor_1_lewo;
      S     #H_Zabierz_do_Nast;
//reset sygn³u zabierz
      AN    #i_Foto_Przod;
      AN    #i_Foto_Tyl;
      A     #Oddanie_Palety;
      =     #Temp_Help_1;
      CALL  #Opuszczenie_Bandy (
           IN                       := #Temp_Help_1,
           PT                       := T#2S,
           Q_0                      := #Temp_Help_2,
           ET                       := #Czas_aktualny);
      A     #Temp_Help_2;
      O;
      AN    #i_Zez_od_Nast;
      R     #H_Zabierz_do_Nast;
      A     #i_Paleta_Dost_Od_Nast;
      FP    #Zbocze_1;
      R     #Help_A_Motor_1_lewo;
      R     #Oddanie_Palety;
      R     #H_Zabierz_do_Nast;
      SET;
//wylacz toggle
      R     #Toggle;
//skocz do koniec
NETWORK
TITLE =
//Resetowanie Startu bindowania gdy bindowanie zalaczone
con:  NOP   0;
NETWORK
TITLE =
//Wrunkowe resetowanie zezwolen
// warunkowy reset zezwolenia
      O     #Help_Motor_2_obr_lewo;
      O     #Help_Motor_2_obr_prawo;
      ON    "Blok_Para".Poz_0_st;
      ON    #i_Bind_Poz_Podst;
      R     #H_Zez_do_Pop;
      R     #H_Zabierz_do_Nast;
NETWORK
TITLE =
//Bindownica
bind: NOP   0;
      CALL  #Bindowanie (
           i_Marka_Bezpieczenstwa   := #i_Marka_Bezpieczenstwa,
           i_Auto_Reczny            := #i_Auto_Reczny,
           i_Bindownica_Auto        := #i_Bindownica_Auto,
           i_Start_Cyklu_Auto       := #H_Start_Cyklu_Bind_Auto,
           i_Reset_Bledu_Cyklu      := #i_Reset_Bledow,
           i_Reset_Cyklu            := #i_Reset_Krokow,
           i_TP_Wiazanie_0_st       := DIX 0.0,
           i_TP_Wiazanie_90_st      := DIX 0.1,
           i_TP_Wiazanie_180_st     := DIX 0.0,
           i_TP_Wiazanie_270_st     := DIX 0.1,
           i_TP_Pozycjonowanie      := DIX 0.2,
           i_s_Zez_Rolki            := DIX 3.0,
           i_Pozycja_Bandy_Lewo     := DIX 1.3,
           i_Pozycja_Bandy_Srodek   := DIX 1.5,
           i_Pozycja_Bandy_Prawo    := DIX 1.4,
           i_Pozycja_Bandy_Potw     := DIX 1.6,
           i_Pozycja_Obr_0st        := DIX 2.3,
           i_Pozycja_Obr_90st       := DIX 2.4,
           i_Pozycja_Obr_180st      := DIX 2.5,
           i_Pozycja_Obr_270st      := DIX 2.6,
           i_Pozycja_Obr_Osiagnieta := DIX 2.7,
           i_Bind_Obwod_Ok          := #i_Bind_Obwod_Ok,
           i_Bind_Poloz_Podst       := "M_Bindownica_Poz_Podst",
           i_Bind_Start_Kon_Wiaz    := #i_Bind_Start_Kon,
           i_Bind_Blad              := #i_Bind_Blad,
           i_Wyjazd_Warunkowy       := DIX 0.6,
           i_Fotokomorki_Pokryte    := #Paleta_rowno_na_stan,
           i_Start_Cyklu_Reczny     := #H_Start_Cyklu_Bind_Recz,
           o_Pozycjonuj_Lewo        := DIX 1.0,
           o_Pozycjonuj_Prawo       := DIX 1.1,
           o_Pozycjonuj_Srodek      := DIX 1.2,
           o_Jedz_Na_0st            := DIX 1.7,
           o_Jedz_Na_90st           := DIX 2.0,
           o_Jedz_Na_180st          := DIX 2.1,
           o_Jedz_Na_270st          := DIX 2.2,
           o_Bind_Zez_Na_Prace      := #Help_B_Zez_Na_Prace,
           o_Bind_Start_Wiazan      := #Help_B_Start_Wiazan,
           o_Koniec_Cyklu           := #Help_Bin_Koniec_Cyklu,
           o_Cykl_W_Trakcie         := #H_Cykl_Bind_Trwa,
           o_Blad_Ogolny            := #Help_B_Blad_Ogolny,
           o_Blad_Cyklu             := #H_Blad_Cyklu,
           io_Step_Counter          := DIW 6);
      A     #H_Start_Cyklu_Bind_Auto;
      R     #H_Start_Cyklu_Bind_Auto;
      A     #H_Start_Cyklu_Bind_Recz;
      R     #H_Start_Cyklu_Bind_Recz;
      AN    #Stop_Czas_Kontrolny;
      A     #i_Reset_Krokow;
      JC    end;
//Resetowanie warunkowe marki cyklu startu 
//Powrot do ominiecia 
NETWORK
TITLE =
//Marka bepieczenstwa Pozycjononwanie
      A     #i_Marka_Bezpieczenstwa;
      A     #H_Cykl_Bind_Trwa;
      O;
      A     #i_Marka_Bezpieczenstwa;
      A     #H_Reset_Srodka;
      =     #H_Marka_Bezp_Poz;
NETWORK
TITLE =
//Pozycjonowanie palety
      CALL  #Pozycjonowanie_Palety (
           i_Marka_Bezpieczenstwa   := #H_Marka_Bezp_Poz,
           i_Auto_Reczny            := TRUE,
           i_Pozycjonuj_Lewo        := DIX 1.0,
           i_Pozycjonuj_Prawo       := DIX 1.1,
           i_Pozycjonuj_Srodek      := DIX 1.2,
           i_Foto_Przod             := #i_Foto_Przod,
           i_Foto_Tyl               := #i_Foto_Tyl,
           s_i_Zez_Na_Rolki         := DIX 3.0,
           i_Czas_Jazdy_Prawo       := T#1S500MS,
           i_Czas_Jazdy_Lewo        := T#1S500MS,
           i_Czas_Opoznienia        := T#1S,
           i_Czas_Powrotu_Prawo     := T#2S,
           i_Czas_Powrotu_Lewo      := T#2S400MS,
           s_i_Blokada_Obrotu       := #Silnik_Rolek_Nie_Pracuje,
           i_Resetuj_Srodek         := #H_Reset_Srodka,
           o_Pozycja_Lewo           := DIX 1.3,
           o_Pozycja_Prawo          := DIX 1.4,
           o_Pozycja_Srodek         := DIX 1.5,
           o_Potw_Pozycji           := DIX 1.6,
           o_Motor_Lewo             := #Help_AP_Motor_1_Lewo,
           o_Motor_Prawo            := #Help_AP_Motor_1_Prawo,
           o_Motor_Wolno            := #Help_AP_Motor_1_Wolno,
           s_o_Zez_Na_Obrot         := DIX 3.1);	//czas pozycjonowania prawo / czas pozycjonowania lewo / czas powrotu od prwej / czas powrotu od lewej
      AN    "Blok_Para".Banda_Poz_Srodek;
      R     #H_Reset_Srodka;
NETWORK
TITLE =
//Marka bezpieczenstwa sterowania obrotu
      A     #i_Marka_Bezpieczenstwa;
      AN    #i_Auto_Reczny;
      AN    #H_Cykl_Bind_Trwa;
      O;
      A     #i_Marka_Bezpieczenstwa;
      A     #H_Cykl_Bind_Trwa;
      O;
      A     #i_Marka_Bezpieczenstwa;
      AN    #H_Cykl_Bind_Trwa;
      A     "Auto_Reczny";
      =     #H_Marka_Bezp_Obr;
      A     #i_Auto_Reczny;
      O;
      A     #H_Cykl_Bind_Trwa;
      =     #H_Auto_Reczny_Ster_Obr;
NETWORK
TITLE =
//Obrot na pozycje 
      CALL  #Sterowanie_Obrotu (
           i_Marka_Bezpieczenstwa   := #H_Marka_Bezp_Obr,
           i_Auto_Reczny            := #H_Auto_Reczny_Ster_Obr,
           Zawsze_True              := #i_Zawsze_True,
           Jedz_Na_0st              := DIX 1.7,
           Jedz_Na_90st             := DIX 2.0,
           Jedz_Na_180st            := DIX 2.1,
           Jedz_Na_270_st           := DIX 2.2,
           Czujnik_0st_1            := #i_czuj_0_st_1,
           Czujnik_0st_2            := #i_czuj_0_st_2,
           Czujnik_90st_1           := #i_czuj_90_st_1,
           Czujnik_90st_2           := #i_czuj_90_st_2,
           Czujnik_180st_1          := #i_Czuj_180_st_1,
           Czujnik_180st_2          := #i_Czuj_180_st_2,
           Czujnik_270st_1          := #i_Czuj_270_st_1,
           Czujnik_270st_2          := #i_Czuj_270_st_2,
           Przycisk_Lewo            := #i_PB_Obr_Lewo,
           Przycisk_Prawo           := #i_PB_Obr_Prawo,
           s_Zez_Na_Obr             := DIX 3.1,
           s_Ramie_Bind_w_Tyle      := #i_Bind_Poz_Podst,
           Na_Pozycji_0st           := DIX 2.3,
           Na_Pozycji_90st          := DIX 2.4,
           Na_Pozycji_180st         := DIX 2.5,
           Na_Pozycji_270st         := DIX 2.6,
           Poz_Osiagnieta           := DIX 2.7,
           s_Zez_Na_Rolki           := DIX 3.0,
           Motor_Wolno              := #Help_Motor_2_Wolno,
           Talerz_w_Lewo            := #Help_Motor_2_obr_lewo,
           Talerz_w_Prawo           := #Help_Motor_2_obr_prawo,
           Pozycja                  := DIW 4);
NETWORK
TITLE =
//Wyzwalanie wyjsc
end:  NOP   0;
NETWORK
TITLE =
//Motor rolki lewo
      A     #i_Marka_Bezpieczenstwa;
      A(;
      A(;
      O     #Help_A_Motor_1_lewo;
      O     #Help_AP_Motor_1_Lewo;
      );
      AN    #Help_H_Motor_1_lewo;
      O;
      A     #Help_H_Motor_1_lewo;
      A     "Blok_Para".Poz_0_st;
      AN    #Help_A_Motor_1_lewo;
      AN    #Help_AP_Motor_1_Lewo;
      );
      A     "Blok_Para".Odblokuj_Rolki;
      A     #i_Bind_Poz_Podst;
      A(;
      O     "Blok_Para".Poz_180_st;
      O     "Blok_Para".Poz_0_st;
      );
      =     #o_Motor_1_lewo;
NETWORK
TITLE = Wiaz wzdluz
//Motor rolki prawo
      A     #i_Marka_Bezpieczenstwa;
      A(;
      A(;
      O     #Help_A_Motor_1_prawo;
      O     #Help_AP_Motor_1_Prawo;
      );
      AN    #Help_H_Motor_1_prawo;
      O;
      A     #Help_H_Motor_1_prawo;
      A     "Blok_Para".Poz_0_st;
      AN    #Help_A_Motor_1_prawo;
      AN    #Help_AP_Motor_1_Prawo;
      );
      A     "Blok_Para".Odblokuj_Rolki;
      A     #i_Bind_Poz_Podst;
      A(;
      O     "Blok_Para".Poz_180_st;
      O     "Blok_Para".Poz_0_st;
      );
      =     #o_Motor_1_prawo;
NETWORK
TITLE =
//motor obrotnica lewo
      A     #i_Marka_Bezpieczenstwa;
      A     #Help_Motor_2_obr_lewo;
      A     #i_Bind_Poz_Podst;
      A     "Blok_Para".Odblokuj_Obrotnice;
      =     #o_Motor_2_obr_s_Lewo;
NETWORK
TITLE =
//motor obrotnica prawo
      A     #i_Marka_Bezpieczenstwa;
      A     #Help_Motor_2_obr_prawo;
      A     #i_Bind_Poz_Podst;
      A     "Blok_Para".Odblokuj_Obrotnice;
      =     #o_Motor_2_obr_s_Prawo;
NETWORK
TITLE =
//motor obrotnica wolno
      A     #Help_Motor_2_Wolno;
      =     #o_Motor_2_Wolno;
NETWORK
TITLE =
//Motor rolki wolno
      O     #Help_A_Motor_1_wolno;
      O     #Help_AP_Motor_1_Wolno;
      =     #o_Motor_1_Wolno;
NETWORK
TITLE =
//zalaczeni wiazarki. Uwaga ze wzgledu na gasnacy sygnal
//      A     #i_Marka_Bezpieczenstwa
      A(;
      O     "Blok_Para".Poz_0_st;
      O     "Blok_Para".Poz_90_st;
      O     "Blok_Para".Poz_180_st;
      O     "Blok_Para".Poz_270_st;
      );
      A     #Help_B_Start_Wiazan;
      =     #o_Bind_Start_Wiazania;
NETWORK
TITLE =
//Zezwolenie na prace bindownicy
      A     #i_Marka_Bezpieczenstwa;
      A     #Help_B_Zez_Na_Prace;
      =     #o_Bind_Zez_Na_Prace;
NETWORK
TITLE =
//Blad ogolny Bindownicy
      A     #Help_B_Blad_Ogolny;
      =     #o_Bind_Blad_Ogolny;
NETWORK
TITLE =
//Blad Cyklu
      A     #H_Blad_Cyklu;
      =     #o_Blad_Cyklu;
NETWORK
TITLE =
//Lampka bindowanie
      A     #o_Bind_Start_Wiazania;
      =     #o_Lampka_Bindowanie;
NETWORK
TITLE =
//Cykl bindowanie trwa
      A     #H_Cykl_Bind_Trwa;
      =     #o_Cykl_Bindowania_Trwa;
NETWORK
TITLE =
//Zezwolenie do poprzedniej 
      A     #H_Zez_do_Pop;
      A     #i_Marka_Bezpieczenstwa;
      =     #o_Zez_do_Pop;
NETWORK
TITLE =
//Zabierz do nast
      A     #H_Zabierz_do_Nast;
      A     #i_Marka_Bezpieczenstwa;
      =     #o_Zabierz_do_Nast;
NETWORK
TITLE =
//Zakonczenie dzialania programu
//
//zakonczenie programu
      BEU;
NETWORK
TITLE = warunkowe przejscie na auto
//Tryb jazdy banda rolkowa po zalaczeniu recznego. Po wejsciu w tryb reczny 
//jezeli 
//sie nic nie robilo to mozna wyjsc i maszyna pracuje dalej. 
//***********************Tryb Rezczny*************************
//************************************************************
hand: NOP   0;
//************************************************
//Pierwsze wejscie to resetuj
      AN    #Toggle;
      JCN   h1;
//tu wpisac kod toggle
h1:   NOP   0;
//*************************************************
//wlacz toggle
      SET;
      S     #Toggle;
//**************************************************
//czyszczenie bitow z automatyki
      SET;
      R     #Help_A_Motor_1_lewo;
      R     #Help_A_Motor_1_prawo;
      R     #Help_A_Motor_1_wolno;
      R     #Pobranie_Wlot;
      R     #Oddanie_Palety;
      R     #H_Zez_do_Pop;
      R     #H_Zabierz_do_Nast;
      R     #H2_Doj_Rolki_Wlot;
      R     #H1_Doj_Rolki_Wlot;
//***************************************************
//Start automatyki w trybie recznym
      A     #i_PB_Cykl_Start;
      FP    #Zbocze_2;
      AN    #H_Cykl_Bind_Trwa;
      A(;
      O(;
      A     "Blok_Para".Poz_0_st;
      A     #Paleta_rowno_na_stan;
      );
      O(;
      A     #i_Foto_Tyl;
      A     "Blok_Para".Poz_180_st;
      );
      );
      S     #H_Reset_Srodka;
      S     #Help_Cykl_Start_Reczny;
      AN    #H_Reset_Srodka;
      A     #Help_Cykl_Start_Reczny;
      S     #H_Start_Cyklu_Bind_Recz;
      R     #Help_Cykl_Start_Reczny;
//jezeli start nie dziala to reset wyrownanie fotkomorek
      A     #i_Reset_Krokow;
      =     #H_Reset_Cyklu_Bind;
      R     #H_Reset_Srodka;
      R     #H_Start_Cyklu_Bind_Recz;
      R     #Help_Cykl_Start_Reczny;
//-
      A     #H_Cykl_Bind_Trwa;
      R     #H_Reset_Srodka;
      R     #H_Start_Cyklu_Bind_Recz;
      R     #Help_Cykl_Start_Reczny;
//********************Jazda Reczna*********************
//ustawienie przyciskow
//jazda do tylu przycisk tyl
      A     #i_Zez_Reczny_Od_Pop;
      A     #i_PB_Jazda_Tyl;
      O;
      AN    #i_Foto_Tyl;
      A(;
      A     #i_PB_Jazda_Tyl;
      AN    #i_PB_Jazda_Przod;
      AN    #Help_H_Motor_1_lewo;
      );
      AN    #H_Cykl_Bind_Trwa;
      =     #Help_H_Motor_1_prawo;
//jazda do przodu
      A     #i_Zez_Reczny_Od_Nast;
      A     #i_PB_Jazda_Przod;
      O;
      AN    #i_Foto_Przod;
      A(;
      A     #i_PB_Jazda_Przod;
      AN    #i_PB_Jazda_Tyl;
      AN    #Help_H_Motor_1_prawo;
      );
      AN    #H_Cykl_Bind_Trwa;
      =     #Help_H_Motor_1_lewo;
//wystawienie zezwolen do innych band wspolpracujacych recznie
//zezwolenie do tylu 
//zezwolenie do poprzedniej
      A     "Blok_Para".Poz_0_st;
      A     "Blok_Para".Odblokuj_Rolki;
      A     #Help_H_Motor_1_lewo;
      A     #o_Motor_1_lewo;
      A     #i_Bind_Poz_Podst;
      AN    #H_Cykl_Bind_Trwa;
      =     #o_Zez_Reczny_do_Pop;
//zezwolenie do nastepnej
      A     "Blok_Para".Poz_0_st;
      A     "Blok_Para".Odblokuj_Rolki;
      A     #Help_H_Motor_1_prawo;
      A     #o_Motor_1_prawo;
      A     #i_Bind_Poz_Podst;
      AN    #H_Cykl_Bind_Trwa;
      =     #o_Zez_Reczny_do_nast;
//skok do dalszej czesc programu
      JU    con;
END_FUNCTION_BLOCK

